	VAR robtarget OpenholeUD_2058 := [[509.33, -12.3, 177.5], [0.183051, 0.683002, 0.683002, -0.183051], [0,0,0,0], [9E9, 9E9, 9E9, 9E9, 9E9, 9E9]];
	VAR robtarget OpenholeUD_2059 := [[505.34, -12.3, 177.76], [0.154444, 0.690034, 0.680633, -0.191674], [0,0,0,0], [9E9, 9E9, 9E9, 9E9, 9E9, 9E9]];
	VAR robtarget OpenholeUD_2060 := [[501.35, -12.3, 178.01], [0.143713, 0.692349, 0.68338, -0.181638], [0,0,0,0], [9E9, 9E9, 9E9, 9E9, 9E9, 9E9]];
	VAR robtarget OpenholeUD_2061 := [[497.36, -12.3, 178.27], [0.132627, 0.694557, 0.686061, -0.17123], [0,0,0,0], [9E9, 9E9, 9E9, 9E9, 9E9, 9E9]];
	VAR robtarget OpenholeUD_2062 := [[493.37, -12.3, 178.53], [0.121195, 0.696643, 0.688661, -0.160454], [0,0,0,0], [9E9, 9E9, 9E9, 9E9, 9E9, 9E9]];
	VAR robtarget OpenholeUD_2063 := [[489.38, -12.3, 178.79], [0.109428, 0.698588, 0.691162, -0.149315], [0,0,0,0], [9E9, 9E9, 9E9, 9E9, 9E9, 9E9]];
	VAR robtarget OpenholeUD_2064 := [[485.38, -12.3, 179.05], [0.097343, 0.700374, 0.693545, -0.137825], [0,0,0,0], [9E9, 9E9, 9E9, 9E9, 9E9, 9E9]];
	VAR robtarget OpenholeUD_2065 := [[481.39, -12.3, 179.31], [0.084958, 0.701984, 0.695791, -0.125996], [0,0,0,0], [9E9, 9E9, 9E9, 9E9, 9E9, 9E9]];
	VAR robtarget OpenholeUD_2066 := [[477.4, -12.3, 179.56], [0.072297, 0.703401, 0.697881, -0.113848], [0,0,0,0], [9E9, 9E9, 9E9, 9E9, 9E9, 9E9]];
	VAR robtarget OpenholeUD_2067 := [[473.41, -12.3, 179.82], [0.059389, 0.704608, 0.699798, -0.101403], [0,0,0,0], [9E9, 9E9, 9E9, 9E9, 9E9, 9E9]];
	VAR robtarget OpenholeUD_2068 := [[469.42, -12.3, 180.08], [0.046265, 0.705592, 0.701523, -0.088688], [0,0,0,0], [9E9, 9E9, 9E9, 9E9, 9E9, 9E9]];
	VAR robtarget OpenholeUD_2069 := [[465.43, -12.3, 180.34], [0.032962, 0.706338, 0.703039, -0.075734], [0,0,0,0], [9E9, 9E9, 9E9, 9E9, 9E9, 9E9]];
	VAR robtarget OpenholeUD_2070 := [[461.43, -12.3, 180.6], [0.019518, 0.706837, 0.704333, -0.062574], [0,0,0,0], [9E9, 9E9, 9E9, 9E9, 9E9, 9E9]];
	VAR robtarget OpenholeUD_2071 := [[457.44, -12.3, 180.86], [0.005975, 0.707082, 0.70539, -0.049249], [0,0,0,0], [9E9, 9E9, 9E9, 9E9, 9E9, 9E9]];
	VAR robtarget OpenholeUD_2072 := [[453.45, -12.3, 181.12], [-0.007623, 0.707066, 0.7062, -0.035797], [0,0,0,0], [9E9, 9E9, 9E9, 9E9, 9E9, 9E9]];
	VAR robtarget OpenholeUD_2073 := [[449.46, -12.3, 181.37], [-0.021231, 0.706788, 0.706756, -0.022263], [0,0,0,0], [9E9, 9E9, 9E9, 9E9, 9E9, 9E9]];
	VAR robtarget OpenholeUD_2074 := [[445.47, -12.3, 181.63], [-0.034805, 0.70625, 0.707053, -0.008691], [0,0,0,0], [9E9, 9E9, 9E9, 9E9, 9E9, 9E9]];
	VAR robtarget OpenholeUD_2075 := [[441.48, -12.3, 181.89], [-0.048298, 0.705455, 0.70709, 0.004875], [0,0,0,0], [9E9, 9E9, 9E9, 9E9, 9E9, 9E9]];
	VAR robtarget OpenholeUD_2076 := [[437.48, -12.3, 182.15], [-0.061667, 0.704413, 0.706868, 0.01839], [0,0,0,0], [9E9, 9E9, 9E9, 9E9, 9E9, 9E9]];
	VAR robtarget OpenholeUD_2077 := [[433.49, -12.3, 182.41], [-0.074872, 0.703132, 0.706391, 0.03181], [0,0,0,0], [9E9, 9E9, 9E9, 9E9, 9E9, 9E9]];
	VAR robtarget OpenholeUD_2078 := [[429.5, -12.3, 182.67], [-0.087873, 0.701626, 0.705667, 0.045095], [0,0,0,0], [9E9, 9E9, 9E9, 9E9, 9E9, 9E9]];
	VAR robtarget OpenholeUD_2079 := [[425.51, -12.3, 182.92], [-0.100635, 0.699909, 0.704707, 0.058204], [0,0,0,0], [9E9, 9E9, 9E9, 9E9, 9E9, 9E9]];
	VAR robtarget OpenholeUD_2080 := [[421.52, -12.3, 183.18], [-0.113126, 0.697999, 0.703523, 0.071103], [0,0,0,0], [9E9, 9E9, 9E9, 9E9, 9E9, 9E9]];
	VAR robtarget OpenholeUD_2081 := [[417.53, -12.3, 183.44], [-0.125319, 0.695913, 0.702128, 0.08376], [0,0,0,0], [9E9, 9E9, 9E9, 9E9, 9E9, 9E9]];
	VAR robtarget OpenholeUD_2082 := [[413.54, -12.3, 183.7], [-0.137192, 0.69367, 0.70054, 0.096145], [0,0,0,0], [9E9, 9E9, 9E9, 9E9, 9E9, 9E9]];
	VAR robtarget OpenholeUD_2083 := [[409.54, -12.3, 183.96], [-0.148726, 0.691289, 0.698774, 0.108235], [0,0,0,0], [9E9, 9E9, 9E9, 9E9, 9E9, 9E9]];
	VAR robtarget OpenholeUD_2084 := [[405.55, -12.3, 184.22], [-0.159905, 0.688789, 0.696848, 0.120011], [0,0,0,0], [9E9, 9E9, 9E9, 9E9, 9E9, 9E9]];
	VAR robtarget OpenholeUD_2085 := [[401.56, -12.3, 184.48], [-0.170721, 0.686188, 0.69478, 0.131455], [0,0,0,0], [9E9, 9E9, 9E9, 9E9, 9E9, 9E9]];
	VAR robtarget OpenholeUD_2086 := [[397.57, -12.3, 184.73], [-0.181166, 0.683505, 0.692588, 0.142556], [0,0,0,0], [9E9, 9E9, 9E9, 9E9, 9E9, 9E9]];
	VAR robtarget OpenholeUD_2087 := [[393.58, -12.3, 184.99], [-0.191237, 0.680756, 0.690288, 0.153306], [0,0,0,0], [9E9, 9E9, 9E9, 9E9, 9E9, 9E9]];
	VAR robtarget OpenholeUD_2088 := [[389.36, -12.3, 185.27], [-0.201475, 0.677796, 0.687759, 0.164279], [0,0,0,0], [9E9, 9E9, 9E9, 9E9, 9E9, 9E9]];
	VAR robtarget OpenholeUD_2089 := [[385.36, -12.3, 185.28], [-0.183051, 0.683002, 0.683002, 0.183051], [0,0,0,0], [9E9, 9E9, 9E9, 9E9, 9E9, 9E9]];
	VAR robtarget OpenholeUD_2090 := [[381.36, -12.3, 185.29], [-0.183051, 0.683002, 0.683002, 0.183051], [0,0,0,0], [9E9, 9E9, 9E9, 9E9, 9E9, 9E9]];
	VAR robtarget OpenholeUD_2091 := [[377.36, -12.3, 185.3], [-0.183051, 0.683002, 0.683002, 0.183051], [0,0,0,0], [9E9, 9E9, 9E9, 9E9, 9E9, 9E9]];
	VAR robtarget OpenholeUD_2092 := [[373.36, -12.3, 185.32], [-0.183051, 0.683002, 0.683002, 0.183051], [0,0,0,0], [9E9, 9E9, 9E9, 9E9, 9E9, 9E9]];
	VAR robtarget OpenholeUD_2093 := [[369.36, -12.3, 185.33], [-0.183051, 0.683002, 0.683002, 0.183051], [0,0,0,0], [9E9, 9E9, 9E9, 9E9, 9E9, 9E9]];
	VAR robtarget OpenholeUD_2094 := [[369.36, -12.3, 185.33], [-0.183051, 0.683002, 0.683002, 0.183051], [0,0,0,0], [9E9, 9E9, 9E9, 9E9, 9E9, 9E9]];
	VAR robtarget OpenholeUD_2095 := [[369.36, -13.5, 184.64], [-0.183051, 0.683002, 0.683002, 0.183051], [0,0,0,0], [9E9, 9E9, 9E9, 9E9, 9E9, 9E9]];
	VAR robtarget OpenholeUD_2096 := [[373.36, -13.5, 184.62], [-0.183051, 0.683002, 0.683002, 0.183051], [0,0,0,0], [9E9, 9E9, 9E9, 9E9, 9E9, 9E9]];
	VAR robtarget OpenholeUD_2097 := [[377.36, -13.5, 184.61], [-0.183051, 0.683002, 0.683002, 0.183051], [0,0,0,0], [9E9, 9E9, 9E9, 9E9, 9E9, 9E9]];
	VAR robtarget OpenholeUD_2098 := [[381.36, -13.5, 184.6], [-0.183051, 0.683002, 0.683002, 0.183051], [0,0,0,0], [9E9, 9E9, 9E9, 9E9, 9E9, 9E9]];
	VAR robtarget OpenholeUD_2099 := [[385.36, -13.5, 184.59], [-0.183051, 0.683002, 0.683002, 0.183051], [0,0,0,0], [9E9, 9E9, 9E9, 9E9, 9E9, 9E9]];
	VAR robtarget OpenholeUD_2100 := [[389.36, -13.5, 184.57], [-0.198088, 0.678794, 0.686931, 0.167708], [0,0,0,0], [9E9, 9E9, 9E9, 9E9, 9E9, 9E9]];
	VAR robtarget OpenholeUD_2101 := [[393.35, -13.5, 184.36], [-0.188336, 0.681564, 0.689367, 0.157396], [0,0,0,0], [9E9, 9E9, 9E9, 9E9, 9E9, 9E9]];
	VAR robtarget OpenholeUD_2102 := [[397.34, -13.5, 184.15], [-0.17821, 0.684281, 0.691716, 0.146726], [0,0,0,0], [9E9, 9E9, 9E9, 9E9, 9E9, 9E9]];
	VAR robtarget OpenholeUD_2103 := [[401.34, -13.5, 183.94], [-0.167712, 0.68693, 0.693963, 0.135702], [0,0,0,0], [9E9, 9E9, 9E9, 9E9, 9E9, 9E9]];
	VAR robtarget OpenholeUD_2104 := [[405.33, -13.5, 183.72], [-0.156844, 0.689493, 0.69609, 0.124331], [0,0,0,0], [9E9, 9E9, 9E9, 9E9, 9E9, 9E9]];
	VAR robtarget OpenholeUD_2105 := [[409.33, -13.5, 183.51], [-0.145614, 0.691951, 0.69808, 0.112626], [0,0,0,0], [9E9, 9E9, 9E9, 9E9, 9E9, 9E9]];
	VAR robtarget OpenholeUD_2106 := [[413.32, -13.5, 183.3], [-0.134032, 0.694288, 0.699914, 0.1006], [0,0,0,0], [9E9, 9E9, 9E9, 9E9, 9E9, 9E9]];
	VAR robtarget OpenholeUD_2107 := [[417.32, -13.5, 183.09], [-0.122114, 0.696483, 0.701575, 0.088273], [0,0,0,0], [9E9, 9E9, 9E9, 9E9, 9E9, 9E9]];
	VAR robtarget OpenholeUD_2108 := [[421.31, -13.5, 182.87], [-0.109878, 0.698518, 0.703046, 0.07567], [0,0,0,0], [9E9, 9E9, 9E9, 9E9, 9E9, 9E9]];
	VAR robtarget OpenholeUD_2109 := [[425.31, -13.5, 182.66], [-0.097347, 0.700374, 0.704311, 0.062816], [0,0,0,0], [9E9, 9E9, 9E9, 9E9, 9E9, 9E9]];
	VAR robtarget OpenholeUD_2110 := [[429.3, -13.5, 182.45], [-0.08455, 0.702034, 0.705355, 0.049744], [0,0,0,0], [9E9, 9E9, 9E9, 9E9, 9E9, 9E9]];
	VAR robtarget OpenholeUD_2111 := [[433.29, -13.5, 182.24], [-0.071518, 0.703481, 0.706165, 0.036489], [0,0,0,0], [9E9, 9E9, 9E9, 9E9, 9E9, 9E9]];
	VAR robtarget OpenholeUD_2112 := [[437.29, -13.5, 182.02], [-0.058286, 0.7047, 0.70673, 0.023089], [0,0,0,0], [9E9, 9E9, 9E9, 9E9, 9E9, 9E9]];
	VAR robtarget OpenholeUD_2113 := [[441.28, -13.5, 181.81], [-0.044894, 0.70568, 0.707042, 0.009586], [0,0,0,0], [9E9, 9E9, 9E9, 9E9, 9E9, 9E9]];
	VAR robtarget OpenholeUD_2114 := [[445.45, -13.5, 181.59], [-0.030809, 0.706435, 0.707092, -0.004555], [0,0,0,0], [9E9, 9E9, 9E9, 9E9, 9E9, 9E9]];
	VAR robtarget OpenholeUD_2115 := [[445.45, -13.5, 181.59], [-0.030809, 0.706435, 0.707092, -0.004555], [0,0,0,0], [9E9, 9E9, 9E9, 9E9, 9E9, 9E9]];
	VAR robtarget OpenholeUD_2116 := [[444.22, -14.7, 181.59], [-0.030884, 0.706432, 0.707097, 0.003667], [0,0,0,0], [9E9, 9E9, 9E9, 9E9, 9E9, 9E9]];
	VAR robtarget OpenholeUD_2117 := [[440.23, -14.7, 181.76], [-0.04439, 0.705712, 0.706897, 0.017215], [0,0,0,0], [9E9, 9E9, 9E9, 9E9, 9E9, 9E9]];
	VAR robtarget OpenholeUD_2118 := [[436.23, -14.7, 181.93], [-0.057772, 0.704743, 0.706441, 0.030684], [0,0,0,0], [9E9, 9E9, 9E9, 9E9, 9E9, 9E9]];
	VAR robtarget OpenholeUD_2119 := [[432.23, -14.7, 182.09], [-0.07099, 0.703534, 0.705735, 0.04403], [0,0,0,0], [9E9, 9E9, 9E9, 9E9, 9E9, 9E9]];
	VAR robtarget OpenholeUD_2120 := [[428.24, -14.7, 182.26], [-0.084005, 0.702099, 0.704788, 0.057215], [0,0,0,0], [9E9, 9E9, 9E9, 9E9, 9E9, 9E9]];
	VAR robtarget OpenholeUD_2121 := [[424.24, -14.7, 182.43], [-0.096783, 0.700452, 0.703613, 0.070201], [0,0,0,0], [9E9, 9E9, 9E9, 9E9, 9E9, 9E9]];
	VAR robtarget OpenholeUD_2122 := [[420.24, -14.7, 182.59], [-0.109291, 0.69861, 0.702224, 0.082953], [0,0,0,0], [9E9, 9E9, 9E9, 9E9, 9E9, 9E9]];
	VAR robtarget OpenholeUD_2123 := [[416.25, -14.7, 182.76], [-0.121503, 0.69659, 0.700636, 0.095443], [0,0,0,0], [9E9, 9E9, 9E9, 9E9, 9E9, 9E9]];
	VAR robtarget OpenholeUD_2124 := [[412.25, -14.7, 182.93], [-0.133395, 0.69441, 0.698865, 0.107643], [0,0,0,0], [9E9, 9E9, 9E9, 9E9, 9E9, 9E9]];
	VAR robtarget OpenholeUD_2125 := [[408.25, -14.7, 183.09], [-0.14495, 0.692091, 0.69693, 0.119534], [0,0,0,0], [9E9, 9E9, 9E9, 9E9, 9E9, 9E9]];
	VAR robtarget OpenholeUD_2126 := [[404.26, -14.7, 183.26], [-0.156153, 0.689649, 0.694848, 0.131096], [0,0,0,0], [9E9, 9E9, 9E9, 9E9, 9E9, 9E9]];
	VAR robtarget OpenholeUD_2127 := [[400.26, -14.7, 183.43], [-0.166993, 0.687105, 0.692637, 0.142317], [0,0,0,0], [9E9, 9E9, 9E9, 9E9, 9E9, 9E9]];
	VAR robtarget OpenholeUD_2128 := [[396.27, -14.7, 183.59], [-0.177464, 0.684475, 0.690315, 0.153186], [0,0,0,0], [9E9, 9E9, 9E9, 9E9, 9E9, 9E9]];
	VAR robtarget OpenholeUD_2129 := [[389.35, -14.7, 183.88], [-0.194694, 0.679775, 0.686085, 0.171135], [0,0,0,0], [9E9, 9E9, 9E9, 9E9, 9E9, 9E9]];
	VAR robtarget OpenholeUD_2130 := [[385.35, -14.7, 183.89], [-0.183051, 0.683002, 0.683002, 0.183051], [0,0,0,0], [9E9, 9E9, 9E9, 9E9, 9E9, 9E9]];
	VAR robtarget OpenholeUD_2131 := [[381.35, -14.7, 183.91], [-0.183051, 0.683002, 0.683002, 0.183051], [0,0,0,0], [9E9, 9E9, 9E9, 9E9, 9E9, 9E9]];
	VAR robtarget OpenholeUD_2132 := [[377.35, -14.7, 183.92], [-0.183051, 0.683002, 0.683002, 0.183051], [0,0,0,0], [9E9, 9E9, 9E9, 9E9, 9E9, 9E9]];
	VAR robtarget OpenholeUD_2133 := [[369.35, -14.7, 183.94], [-0.183051, 0.683002, 0.683002, 0.183051], [0,0,0,0], [9E9, 9E9, 9E9, 9E9, 9E9, 9E9]];
	VAR robtarget OpenholeUD_2134 := [[369.35, -14.7, 183.94], [-0.183051, 0.683002, 0.683002, 0.183051], [0,0,0,0], [9E9, 9E9, 9E9, 9E9, 9E9, 9E9]];
	VAR robtarget OpenholeUD_2135 := [[369.35, -15.9, 183.25], [-0.183051, 0.683002, 0.683002, 0.183051], [0,0,0,0], [9E9, 9E9, 9E9, 9E9, 9E9, 9E9]];
	VAR robtarget OpenholeUD_2136 := [[373.35, -15.9, 183.24], [-0.183051, 0.683002, 0.683002, 0.183051], [0,0,0,0], [9E9, 9E9, 9E9, 9E9, 9E9, 9E9]];
	VAR robtarget OpenholeUD_2137 := [[377.35, -15.9, 183.22], [-0.183051, 0.683002, 0.683002, 0.183051], [0,0,0,0], [9E9, 9E9, 9E9, 9E9, 9E9, 9E9]];
	VAR robtarget OpenholeUD_2138 := [[381.35, -15.9, 183.21], [-0.183051, 0.683002, 0.683002, 0.183051], [0,0,0,0], [9E9, 9E9, 9E9, 9E9, 9E9, 9E9]];
	VAR robtarget OpenholeUD_2139 := [[389.35, -15.9, 183.19], [-0.191292, 0.68074, 0.685222, 0.174561], [0,0,0,0], [9E9, 9E9, 9E9, 9E9, 9E9, 9E9]];
	VAR robtarget OpenholeUD_2140 := [[393.35, -15.9, 183.07], [-0.181391, 0.683445, 0.687735, 0.164377], [0,0,0,0], [9E9, 9E9, 9E9, 9E9, 9E9, 9E9]];
	VAR robtarget OpenholeUD_2141 := [[397.35, -15.9, 182.95], [-0.171117, 0.68609, 0.690171, 0.153832], [0,0,0,0], [9E9, 9E9, 9E9, 9E9, 9E9, 9E9]];
	VAR robtarget OpenholeUD_2142 := [[401.35, -15.9, 182.83], [-0.160474, 0.688657, 0.692511, 0.142928], [0,0,0,0], [9E9, 9E9, 9E9, 9E9, 9E9, 9E9]];
	VAR robtarget OpenholeUD_2143 := [[405.34, -15.9, 182.71], [-0.149465, 0.69113, 0.694739, 0.131672], [0,0,0,0], [9E9, 9E9, 9E9, 9E9, 9E9, 9E9]];
	VAR robtarget OpenholeUD_2144 := [[409.34, -15.9, 182.59], [-0.138098, 0.69349, 0.696837, 0.120075], [0,0,0,0], [9E9, 9E9, 9E9, 9E9, 9E9, 9E9]];
	VAR robtarget OpenholeUD_2145 := [[413.34, -15.9, 182.46], [-0.126386, 0.69572, 0.698787, 0.108151], [0,0,0,0], [9E9, 9E9, 9E9, 9E9, 9E9, 9E9]];
	VAR robtarget OpenholeUD_2146 := [[417.34, -15.9, 182.34], [-0.114345, 0.6978, 0.700571, 0.095917], [0,0,0,0], [9E9, 9E9, 9E9, 9E9, 9E9, 9E9]];
	VAR robtarget OpenholeUD_2147 := [[421.34, -15.9, 182.22], [-0.101994, 0.699712, 0.702172, 0.083396], [0,0,0,0], [9E9, 9E9, 9E9, 9E9, 9E9, 9E9]];
	VAR robtarget OpenholeUD_2148 := [[425.34, -15.9, 182.1], [-0.089359, 0.701438, 0.703572, 0.070615], [0,0,0,0], [9E9, 9E9, 9E9, 9E9, 9E9, 9E9]];
	VAR robtarget OpenholeUD_2149 := [[429.33, -15.9, 181.98], [-0.076469, 0.70296, 0.704757, 0.057603], [0,0,0,0], [9E9, 9E9, 9E9, 9E9, 9E9, 9E9]];
	VAR robtarget OpenholeUD_2150 := [[433.33, -15.9, 181.86], [-0.063356, 0.704263, 0.705712, 0.044396], [0,0,0,0], [9E9, 9E9, 9E9, 9E9, 9E9, 9E9]];
	VAR robtarget OpenholeUD_2151 := [[437.33, -15.9, 181.74], [-0.050056, 0.705333, 0.706426, 0.031031], [0,0,0,0], [9E9, 9E9, 9E9, 9E9, 9E9, 9E9]];
	VAR robtarget OpenholeUD_2152 := [[443.48, -15.9, 181.56], [-0.029327, 0.706498, 0.707032, 0.010255], [0,0,0,0], [9E9, 9E9, 9E9, 9E9, 9E9, 9E9]];
	VAR robtarget OpenholeUD_2153 := [[443.48, -15.9, 181.56], [-0.029327, 0.706498, 0.707032, 0.010255], [0,0,0,0], [9E9, 9E9, 9E9, 9E9, 9E9, 9E9]];
	VAR robtarget OpenholeUD_2154 := [[443.05, -17.1, 181.5], [-0.026721, 0.706602, 0.70693, 0.015795], [0,0,0,0], [9E9, 9E9, 9E9, 9E9, 9E9, 9E9]];
	VAR robtarget OpenholeUD_2155 := [[439.05, -17.1, 181.57], [-0.040236, 0.705961, 0.706499, 0.029304], [0,0,0,0], [9E9, 9E9, 9E9, 9E9, 9E9, 9E9]];
	VAR robtarget OpenholeUD_2156 := [[435.05, -17.1, 181.65], [-0.053629, 0.70507, 0.705816, 0.042707], [0,0,0,0], [9E9, 9E9, 9E9, 9E9, 9E9, 9E9]];
	VAR robtarget OpenholeUD_2157 := [[431.05, -17.1, 181.72], [-0.066861, 0.703939, 0.704889, 0.055961], [0,0,0,0], [9E9, 9E9, 9E9, 9E9, 9E9, 9E9]];
	VAR robtarget OpenholeUD_2158 := [[427.05, -17.1, 181.79], [-0.079891, 0.702579, 0.703729, 0.069029], [0,0,0,0], [9E9, 9E9, 9E9, 9E9, 9E9, 9E9]];
	VAR robtarget OpenholeUD_2159 := [[423.05, -17.1, 181.87], [-0.092685, 0.701006, 0.702351, 0.081875], [0,0,0,0], [9E9, 9E9, 9E9, 9E9, 9E9, 9E9]];
	VAR robtarget OpenholeUD_2160 := [[419.05, -17.1, 181.94], [-0.105212, 0.699236, 0.700768, 0.094468], [0,0,0,0], [9E9, 9E9, 9E9, 9E9, 9E9, 9E9]];
	VAR robtarget OpenholeUD_2161 := [[415.05, -17.1, 182.02], [-0.117445, 0.697285, 0.698998, 0.106779], [0,0,0,0], [9E9, 9E9, 9E9, 9E9, 9E9, 9E9]];
	VAR robtarget OpenholeUD_2162 := [[411.05, -17.1, 182.09], [-0.12936, 0.695173, 0.697058, 0.118786], [0,0,0,0], [9E9, 9E9, 9E9, 9E9, 9E9, 9E9]];
	VAR robtarget OpenholeUD_2163 := [[407.05, -17.1, 182.17], [-0.14094, 0.692918, 0.694966, 0.130469], [0,0,0,0], [9E9, 9E9, 9E9, 9E9, 9E9, 9E9]];
	VAR robtarget OpenholeUD_2164 := [[403.05, -17.1, 182.24], [-0.15217, 0.690539, 0.69274, 0.141813], [0,0,0,0], [9E9, 9E9, 9E9, 9E9, 9E9, 9E9]];
	VAR robtarget OpenholeUD_2165 := [[399.05, -17.1, 182.31], [-0.163039, 0.688054, 0.690399, 0.152806], [0,0,0,0], [9E9, 9E9, 9E9, 9E9, 9E9, 9E9]];
	VAR robtarget OpenholeUD_2166 := [[395.06, -17.1, 182.39], [-0.173542, 0.68548, 0.687959, 0.16344], [0,0,0,0], [9E9, 9E9, 9E9, 9E9, 9E9, 9E9]];
	VAR robtarget OpenholeUD_2167 := [[389.35, -17.1, 182.49], [-0.187884, 0.681689, 0.68434, 0.177984], [0,0,0,0], [9E9, 9E9, 9E9, 9E9, 9E9, 9E9]];
	VAR robtarget OpenholeUD_2168 := [[385.35, -17.1, 182.51], [-0.183051, 0.683002, 0.683002, 0.183051], [0,0,0,0], [9E9, 9E9, 9E9, 9E9, 9E9, 9E9]];
	VAR robtarget OpenholeUD_2169 := [[381.35, -17.1, 182.52], [-0.183051, 0.683002, 0.683002, 0.183051], [0,0,0,0], [9E9, 9E9, 9E9, 9E9, 9E9, 9E9]];
	VAR robtarget OpenholeUD_2170 := [[377.35, -17.1, 182.53], [-0.183051, 0.683002, 0.683002, 0.183051], [0,0,0,0], [9E9, 9E9, 9E9, 9E9, 9E9, 9E9]];
	VAR robtarget OpenholeUD_2171 := [[369.35, -17.1, 182.56], [-0.183051, 0.683002, 0.683002, 0.183051], [0,0,0,0], [9E9, 9E9, 9E9, 9E9, 9E9, 9E9]];
	VAR robtarget OpenholeUD_2172 := [[369.35, -17.1, 182.56], [-0.183051, 0.683002, 0.683002, 0.183051], [0,0,0,0], [9E9, 9E9, 9E9, 9E9, 9E9, 9E9]];
	VAR robtarget OpenholeUD_2173 := [[369.35, -18.3, 181.86], [-0.183051, 0.683002, 0.683002, 0.183051], [0,0,0,0], [9E9, 9E9, 9E9, 9E9, 9E9, 9E9]];
	VAR robtarget OpenholeUD_2174 := [[373.35, -18.3, 181.85], [-0.183051, 0.683002, 0.683002, 0.183051], [0,0,0,0], [9E9, 9E9, 9E9, 9E9, 9E9, 9E9]];
	VAR robtarget OpenholeUD_2175 := [[377.35, -18.3, 181.84], [-0.183051, 0.683002, 0.683002, 0.183051], [0,0,0,0], [9E9, 9E9, 9E9, 9E9, 9E9, 9E9]];
	VAR robtarget OpenholeUD_2176 := [[381.35, -18.3, 181.83], [-0.183051, 0.683002, 0.683002, 0.183051], [0,0,0,0], [9E9, 9E9, 9E9, 9E9, 9E9, 9E9]];
	VAR robtarget OpenholeUD_2177 := [[385.35, -18.3, 181.81], [-0.183051, 0.683002, 0.683002, 0.183051], [0,0,0,0], [9E9, 9E9, 9E9, 9E9, 9E9, 9E9]];
	VAR robtarget OpenholeUD_2178 := [[389.35, -18.3, 181.8], [-0.18447, 0.682621, 0.683442, 0.181403], [0,0,0,0], [9E9, 9E9, 9E9, 9E9, 9E9, 9E9]];
	VAR robtarget OpenholeUD_2179 := [[393.35, -18.3, 181.77], [-0.174424, 0.685256, 0.68603, 0.171354], [0,0,0,0], [9E9, 9E9, 9E9, 9E9, 9E9, 9E9]];
	VAR robtarget OpenholeUD_2180 := [[397.35, -18.3, 181.74], [-0.164009, 0.687823, 0.688548, 0.160941], [0,0,0,0], [9E9, 9E9, 9E9, 9E9, 9E9, 9E9]];
	VAR robtarget OpenholeUD_2181 := [[401.35, -18.3, 181.72], [-0.153227, 0.690305, 0.690978, 0.150165], [0,0,0,0], [9E9, 9E9, 9E9, 9E9, 9E9, 9E9]];
	VAR robtarget OpenholeUD_2182 := [[405.35, -18.3, 181.69], [-0.142084, 0.692685, 0.693304, 0.139032], [0,0,0,0], [9E9, 9E9, 9E9, 9E9, 9E9, 9E9]];
	VAR robtarget OpenholeUD_2183 := [[409.35, -18.3, 181.66], [-0.130588, 0.694944, 0.695507, 0.127552], [0,0,0,0], [9E9, 9E9, 9E9, 9E9, 9E9, 9E9]];
	VAR robtarget OpenholeUD_2184 := [[413.35, -18.3, 181.63], [-0.118754, 0.697064, 0.697571, 0.115737], [0,0,0,0], [9E9, 9E9, 9E9, 9E9, 9E9, 9E9]];
	VAR robtarget OpenholeUD_2185 := [[417.35, -18.3, 181.61], [-0.106598, 0.699026, 0.699476, 0.103605], [0,0,0,0], [9E9, 9E9, 9E9, 9E9, 9E9, 9E9]];
	VAR robtarget OpenholeUD_2186 := [[421.35, -18.3, 181.58], [-0.094141, 0.700812, 0.701204, 0.091176], [0,0,0,0], [9E9, 9E9, 9E9, 9E9, 9E9, 9E9]];
	VAR robtarget OpenholeUD_2187 := [[425.35, -18.3, 181.55], [-0.081411, 0.702405, 0.702739, 0.078477], [0,0,0,0], [9E9, 9E9, 9E9, 9E9, 9E9, 9E9]];
	VAR robtarget OpenholeUD_2188 := [[429.35, -18.3, 181.52], [-0.068436, 0.703787, 0.704063, 0.065535], [0,0,0,0], [9E9, 9E9, 9E9, 9E9, 9E9, 9E9]];
	VAR robtarget OpenholeUD_2189 := [[433.35, -18.3, 181.49], [-0.055252, 0.704945, 0.705164, 0.052386], [0,0,0,0], [9E9, 9E9, 9E9, 9E9, 9E9, 9E9]];
	VAR robtarget OpenholeUD_2190 := [[437.35, -18.3, 181.47], [-0.041895, 0.705865, 0.706027, 0.039065], [0,0,0,0], [9E9, 9E9, 9E9, 9E9, 9E9, 9E9]];
	VAR robtarget OpenholeUD_2191 := [[442.86, -18.3, 181.43], [-0.023279, 0.706723, 0.70681, 0.0205], [0,0,0,0], [9E9, 9E9, 9E9, 9E9, 9E9, 9E9]];
	VAR robtarget OpenholeUD_2192 := [[442.86, -18.3, 181.43], [-0.023279, 0.706723, 0.70681, 0.0205], [0,0,0,0], [9E9, 9E9, 9E9, 9E9, 9E9, 9E9]];
	VAR robtarget OpenholeUD_2193 := [[442.9, -19.5, 181.35], [-0.019074, 0.706849, 0.706684, 0.024443], [0,0,0,0], [9E9, 9E9, 9E9, 9E9, 9E9, 9E9]];
	VAR robtarget OpenholeUD_2194 := [[438.9, -19.5, 181.33], [-0.032618, 0.706354, 0.706089, 0.037919], [0,0,0,0], [9E9, 9E9, 9E9, 9E9, 9E9, 9E9]];
	VAR robtarget OpenholeUD_2195 := [[434.9, -19.5, 181.32], [-0.046054, 0.705605, 0.705245, 0.051273], [0,0,0,0], [9E9, 9E9, 9E9, 9E9, 9E9, 9E9]];
	VAR robtarget OpenholeUD_2196 := [[430.9, -19.5, 181.3], [-0.059339, 0.704613, 0.704162, 0.064463], [0,0,0,0], [9E9, 9E9, 9E9, 9E9, 9E9, 9E9]];
	VAR robtarget OpenholeUD_2197 := [[426.9, -19.5, 181.28], [-0.072435, 0.703387, 0.702852, 0.077453], [0,0,0,0], [9E9, 9E9, 9E9, 9E9, 9E9, 9E9]];
	VAR robtarget OpenholeUD_2198 := [[422.9, -19.5, 181.26], [-0.085306, 0.701942, 0.701329, 0.090208], [0,0,0,0], [9E9, 9E9, 9E9, 9E9, 9E9, 9E9]];
	VAR robtarget OpenholeUD_2199 := [[418.9, -19.5, 181.24], [-0.09792, 0.700294, 0.699609, 0.102697], [0,0,0,0], [9E9, 9E9, 9E9, 9E9, 9E9, 9E9]];
	VAR robtarget OpenholeUD_2200 := [[414.9, -19.5, 181.22], [-0.110247, 0.698459, 0.69771, 0.114895], [0,0,0,0], [9E9, 9E9, 9E9, 9E9, 9E9, 9E9]];
	VAR robtarget OpenholeUD_2201 := [[410.9, -19.5, 181.21], [-0.122265, 0.696456, 0.695649, 0.126778], [0,0,0,0], [9E9, 9E9, 9E9, 9E9, 9E9, 9E9]];
	VAR robtarget OpenholeUD_2202 := [[406.9, -19.5, 181.19], [-0.133955, 0.694303, 0.693444, 0.138329], [0,0,0,0], [9E9, 9E9, 9E9, 9E9, 9E9, 9E9]];
	VAR robtarget OpenholeUD_2203 := [[402.9, -19.5, 181.17], [-0.145299, 0.692017, 0.691115, 0.149535], [0,0,0,0], [9E9, 9E9, 9E9, 9E9, 9E9, 9E9]];
	VAR robtarget OpenholeUD_2204 := [[398.9, -19.5, 181.15], [-0.156289, 0.689619, 0.688678, 0.160384], [0,0,0,0], [9E9, 9E9, 9E9, 9E9, 9E9, 9E9]];
	VAR robtarget OpenholeUD_2205 := [[394.9, -19.5, 181.13], [-0.166914, 0.687124, 0.686151, 0.170871], [0,0,0,0], [9E9, 9E9, 9E9, 9E9, 9E9, 9E9]];
	VAR robtarget OpenholeUD_2206 := [[389.35, -19.5, 181.11], [-0.181051, 0.683535, 0.682526, 0.184819], [0,0,0,0], [9E9, 9E9, 9E9, 9E9, 9E9, 9E9]];
	VAR robtarget OpenholeUD_2207 := [[385.35, -19.5, 181.12], [-0.183051, 0.683002, 0.683002, 0.183051], [0,0,0,0], [9E9, 9E9, 9E9, 9E9, 9E9, 9E9]];
	VAR robtarget OpenholeUD_2208 := [[381.35, -19.5, 181.13], [-0.183051, 0.683002, 0.683002, 0.183051], [0,0,0,0], [9E9, 9E9, 9E9, 9E9, 9E9, 9E9]];
	VAR robtarget OpenholeUD_2209 := [[377.35, -19.5, 181.15], [-0.183051, 0.683002, 0.683002, 0.183051], [0,0,0,0], [9E9, 9E9, 9E9, 9E9, 9E9, 9E9]];
	VAR robtarget OpenholeUD_2210 := [[373.35, -19.5, 181.16], [-0.183051, 0.683002, 0.683002, 0.183051], [0,0,0,0], [9E9, 9E9, 9E9, 9E9, 9E9, 9E9]];
	VAR robtarget OpenholeUD_2211 := [[369.35, -19.5, 181.17], [-0.183051, 0.683002, 0.683002, 0.183051], [0,0,0,0], [9E9, 9E9, 9E9, 9E9, 9E9, 9E9]];
	VAR robtarget OpenholeUD_2212 := [[369.35, -19.5, 181.17], [-0.183051, 0.683002, 0.683002, 0.183051], [0,0,0,0], [9E9, 9E9, 9E9, 9E9, 9E9, 9E9]];
	VAR robtarget OpenholeUD_2213 := [[369.34, -20.7, 180.48], [-0.183051, 0.683002, 0.683002, 0.183051], [0,0,0,0], [9E9, 9E9, 9E9, 9E9, 9E9, 9E9]];
	VAR robtarget OpenholeUD_2214 := [[373.34, -20.7, 180.47], [-0.183051, 0.683002, 0.683002, 0.183051], [0,0,0,0], [9E9, 9E9, 9E9, 9E9, 9E9, 9E9]];
	VAR robtarget OpenholeUD_2215 := [[377.34, -20.7, 180.45], [-0.183051, 0.683002, 0.683002, 0.183051], [0,0,0,0], [9E9, 9E9, 9E9, 9E9, 9E9, 9E9]];
	VAR robtarget OpenholeUD_2216 := [[381.34, -20.7, 180.44], [-0.183051, 0.683002, 0.683002, 0.183051], [0,0,0,0], [9E9, 9E9, 9E9, 9E9, 9E9, 9E9]];
	VAR robtarget OpenholeUD_2217 := [[385.34, -20.7, 180.43], [-0.183051, 0.683002, 0.683002, 0.183051], [0,0,0,0], [9E9, 9E9, 9E9, 9E9, 9E9, 9E9]];
	VAR robtarget OpenholeUD_2218 := [[389.34, -20.7, 180.41], [-0.177628, 0.684433, 0.681594, 0.188229], [0,0,0,0], [9E9, 9E9, 9E9, 9E9, 9E9, 9E9]];
	VAR robtarget OpenholeUD_2219 := [[393.34, -20.7, 180.48], [-0.167444, 0.686995, 0.684253, 0.178321], [0,0,0,0], [9E9, 9E9, 9E9, 9E9, 9E9, 9E9]];
	VAR robtarget OpenholeUD_2220 := [[397.34, -20.7, 180.54], [-0.156894, 0.689481, 0.686848, 0.168045], [0,0,0,0], [9E9, 9E9, 9E9, 9E9, 9E9, 9E9]];
	VAR robtarget OpenholeUD_2221 := [[401.34, -20.7, 180.61], [-0.14598, 0.691874, 0.689365, 0.157404], [0,0,0,0], [9E9, 9E9, 9E9, 9E9, 9E9, 9E9]];
	VAR robtarget OpenholeUD_2222 := [[405.34, -20.7, 180.67], [-0.134709, 0.694157, 0.691785, 0.146401], [0,0,0,0], [9E9, 9E9, 9E9, 9E9, 9E9, 9E9]];
	VAR robtarget OpenholeUD_2223 := [[409.34, -20.7, 180.74], [-0.123092, 0.69631, 0.694091, 0.135046], [0,0,0,0], [9E9, 9E9, 9E9, 9E9, 9E9, 9E9]];
	VAR robtarget OpenholeUD_2224 := [[413.34, -20.7, 180.8], [-0.111144, 0.698317, 0.696265, 0.12335], [0,0,0,0], [9E9, 9E9, 9E9, 9E9, 9E9, 9E9]];
	VAR robtarget OpenholeUD_2225 := [[417.34, -20.7, 180.87], [-0.098881, 0.700159, 0.698288, 0.111328], [0,0,0,0], [9E9, 9E9, 9E9, 9E9, 9E9, 9E9]];
	VAR robtarget OpenholeUD_2226 := [[421.34, -20.7, 180.93], [-0.086329, 0.701817, 0.700142, 0.099001], [0,0,0,0], [9E9, 9E9, 9E9, 9E9, 9E9, 9E9]];
	VAR robtarget OpenholeUD_2227 := [[425.34, -20.7, 180.99], [-0.073512, 0.703275, 0.701809, 0.086392], [0,0,0,0], [9E9, 9E9, 9E9, 9E9, 9E9, 9E9]];
	VAR robtarget OpenholeUD_2228 := [[429.34, -20.7, 181.06], [-0.060463, 0.704517, 0.703273, 0.073531], [0,0,0,0], [9E9, 9E9, 9E9, 9E9, 9E9, 9E9]];
	VAR robtarget OpenholeUD_2229 := [[433.34, -20.7, 181.12], [-0.047217, 0.705529, 0.704518, 0.060449], [0,0,0,0], [9E9, 9E9, 9E9, 9E9, 9E9, 9E9]];
	VAR robtarget OpenholeUD_2230 := [[437.34, -20.7, 181.19], [-0.033812, 0.706298, 0.705531, 0.047182], [0,0,0,0], [9E9, 9E9, 9E9, 9E9, 9E9, 9E9]];
	VAR robtarget OpenholeUD_2231 := [[443.16, -20.7, 181.28], [-0.014092, 0.706966, 0.706567, 0.027613], [0,0,0,0], [9E9, 9E9, 9E9, 9E9, 9E9, 9E9]];
	VAR robtarget OpenholeUD_2232 := [[443.16, -20.7, 181.28], [-0.014092, 0.706966, 0.706567, 0.027613], [0,0,0,0], [9E9, 9E9, 9E9, 9E9, 9E9, 9E9]];
	VAR robtarget OpenholeUD_2233 := [[443.69, -21.9, 181.22], [-0.00822, 0.707059, 0.706474, 0.029897], [0,0,0,0], [9E9, 9E9, 9E9, 9E9, 9E9, 9E9]];
	VAR robtarget OpenholeUD_2234 := [[439.69, -21.9, 181.11], [-0.021801, 0.706771, 0.705776, 0.043357], [0,0,0,0], [9E9, 9E9, 9E9, 9E9, 9E9, 9E9]];
	VAR robtarget OpenholeUD_2235 := [[435.69, -21.9, 181], [-0.035297, 0.706225, 0.704831, 0.056689], [0,0,0,0], [9E9, 9E9, 9E9, 9E9, 9E9, 9E9]];
	VAR robtarget OpenholeUD_2236 := [[431.69, -21.9, 180.89], [-0.048665, 0.70543, 0.703648, 0.069851], [0,0,0,0], [9E9, 9E9, 9E9, 9E9, 9E9, 9E9]];
	VAR robtarget OpenholeUD_2237 := [[427.69, -21.9, 180.78], [-0.061865, 0.704395, 0.702241, 0.082808], [0,0,0,0], [9E9, 9E9, 9E9, 9E9, 9E9, 9E9]];
	VAR robtarget OpenholeUD_2238 := [[423.7, -21.9, 180.67], [-0.074859, 0.703133, 0.700625, 0.095524], [0,0,0,0], [9E9, 9E9, 9E9, 9E9, 9E9, 9E9]];
	VAR robtarget OpenholeUD_2239 := [[419.7, -21.9, 180.56], [-0.087613, 0.701658, 0.698815, 0.10797], [0,0,0,0], [9E9, 9E9, 9E9, 9E9, 9E9, 9E9]];
	VAR robtarget OpenholeUD_2240 := [[415.7, -21.9, 180.45], [-0.100097, 0.699986, 0.696829, 0.12012], [0,0,0,0], [9E9, 9E9, 9E9, 9E9, 9E9, 9E9]];
	VAR robtarget OpenholeUD_2241 := [[411.7, -21.9, 180.34], [-0.112285, 0.698135, 0.694686, 0.131951], [0,0,0,0], [9E9, 9E9, 9E9, 9E9, 9E9, 9E9]];
	VAR robtarget OpenholeUD_2242 := [[407.7, -21.9, 180.23], [-0.124156, 0.696122, 0.692404, 0.143446], [0,0,0,0], [9E9, 9E9, 9E9, 9E9, 9E9, 9E9]];
	VAR robtarget OpenholeUD_2243 := [[403.7, -21.9, 180.12], [-0.135692, 0.693965, 0.690001, 0.154592], [0,0,0,0], [9E9, 9E9, 9E9, 9E9, 9E9, 9E9]];
	VAR robtarget OpenholeUD_2244 := [[399.7, -21.9, 180.01], [-0.14688, 0.691684, 0.687495, 0.165379], [0,0,0,0], [9E9, 9E9, 9E9, 9E9, 9E9, 9E9]];
	VAR robtarget OpenholeUD_2245 := [[395.71, -21.9, 179.9], [-0.157711, 0.689295, 0.684904, 0.175801], [0,0,0,0], [9E9, 9E9, 9E9, 9E9, 9E9, 9E9]];
	VAR robtarget OpenholeUD_2246 := [[389.34, -21.9, 179.72], [-0.174202, 0.685313, 0.680644, 0.191634], [0,0,0,0], [9E9, 9E9, 9E9, 9E9, 9E9, 9E9]];
	VAR robtarget OpenholeUD_2247 := [[385.34, -21.9, 179.73], [-0.183051, 0.683002, 0.683002, 0.183051], [0,0,0,0], [9E9, 9E9, 9E9, 9E9, 9E9, 9E9]];
	VAR robtarget OpenholeUD_2248 := [[381.34, -21.9, 179.75], [-0.183051, 0.683002, 0.683002, 0.183051], [0,0,0,0], [9E9, 9E9, 9E9, 9E9, 9E9, 9E9]];
	VAR robtarget OpenholeUD_2249 := [[377.34, -21.9, 179.76], [-0.183051, 0.683002, 0.683002, 0.183051], [0,0,0,0], [9E9, 9E9, 9E9, 9E9, 9E9, 9E9]];
	VAR robtarget OpenholeUD_2250 := [[373.34, -21.9, 179.77], [-0.183051, 0.683002, 0.683002, 0.183051], [0,0,0,0], [9E9, 9E9, 9E9, 9E9, 9E9, 9E9]];
	VAR robtarget OpenholeUD_2251 := [[369.34, -21.9, 179.78], [-0.183051, 0.683002, 0.683002, 0.183051], [0,0,0,0], [9E9, 9E9, 9E9, 9E9, 9E9, 9E9]];
	VAR robtarget OpenholeUD_2252 := [[369.34, -21.9, 179.78], [-0.183051, 0.683002, 0.683002, 0.183051], [0,0,0,0], [9E9, 9E9, 9E9, 9E9, 9E9, 9E9]];
	VAR robtarget OpenholeUD_2253 := [[369.34, -23.1, 179.09], [-0.183051, 0.683002, 0.683002, 0.183051], [0,0,0,0], [9E9, 9E9, 9E9, 9E9, 9E9, 9E9]];
	VAR robtarget OpenholeUD_2254 := [[373.34, -23.1, 179.08], [-0.183051, 0.683002, 0.683002, 0.183051], [0,0,0,0], [9E9, 9E9, 9E9, 9E9, 9E9, 9E9]];
	VAR robtarget OpenholeUD_2255 := [[377.34, -23.1, 179.07], [-0.183051, 0.683002, 0.683002, 0.183051], [0,0,0,0], [9E9, 9E9, 9E9, 9E9, 9E9, 9E9]];
	VAR robtarget OpenholeUD_2256 := [[381.34, -23.1, 179.05], [-0.183051, 0.683002, 0.683002, 0.183051], [0,0,0,0], [9E9, 9E9, 9E9, 9E9, 9E9, 9E9]];
	VAR robtarget OpenholeUD_2257 := [[385.34, -23.1, 179.04], [-0.183051, 0.683002, 0.683002, 0.183051], [0,0,0,0], [9E9, 9E9, 9E9, 9E9, 9E9, 9E9]];
	VAR robtarget OpenholeUD_2258 := [[389.34, -23.1, 179.03], [-0.170773, 0.686175, 0.679678, 0.195032], [0,0,0,0], [9E9, 9E9, 9E9, 9E9, 9E9, 9E9]];
	VAR robtarget OpenholeUD_2259 := [[393.34, -23.1, 179.19], [-0.160457, 0.688661, 0.682404, 0.18527], [0,0,0,0], [9E9, 9E9, 9E9, 9E9, 9E9, 9E9]];
	VAR robtarget OpenholeUD_2260 := [[397.33, -23.1, 179.34], [-0.149778, 0.691062, 0.685074, 0.175138], [0,0,0,0], [9E9, 9E9, 9E9, 9E9, 9E9, 9E9]];
	VAR robtarget OpenholeUD_2261 := [[401.33, -23.1, 179.5], [-0.138739, 0.693362, 0.687673, 0.164638], [0,0,0,0], [9E9, 9E9, 9E9, 9E9, 9E9, 9E9]];
	VAR robtarget OpenholeUD_2262 := [[405.33, -23.1, 179.66], [-0.127349, 0.695544, 0.690184, 0.153773], [0,0,0,0], [9E9, 9E9, 9E9, 9E9, 9E9, 9E9]];
	VAR robtarget OpenholeUD_2263 := [[409.32, -23.1, 179.81], [-0.115619, 0.69759, 0.692589, 0.14255], [0,0,0,0], [9E9, 9E9, 9E9, 9E9, 9E9, 9E9]];
	VAR robtarget OpenholeUD_2264 := [[413.32, -23.1, 179.97], [-0.103565, 0.699481, 0.69487, 0.13098], [0,0,0,0], [9E9, 9E9, 9E9, 9E9, 9E9, 9E9]];
	VAR robtarget OpenholeUD_2265 := [[417.32, -23.1, 180.13], [-0.091206, 0.7012, 0.697008, 0.119077], [0,0,0,0], [9E9, 9E9, 9E9, 9E9, 9E9, 9E9]];
	VAR robtarget OpenholeUD_2266 := [[421.31, -23.1, 180.28], [-0.078566, 0.702729, 0.698986, 0.10686], [0,0,0,0], [9E9, 9E9, 9E9, 9E9, 9E9, 9E9]];
	VAR robtarget OpenholeUD_2267 := [[425.31, -23.1, 180.44], [-0.065673, 0.70405, 0.700784, 0.094351], [0,0,0,0], [9E9, 9E9, 9E9, 9E9, 9E9, 9E9]];
	VAR robtarget OpenholeUD_2268 := [[429.31, -23.1, 180.6], [-0.05256, 0.705151, 0.702385, 0.081579], [0,0,0,0], [9E9, 9E9, 9E9, 9E9, 9E9, 9E9]];
	VAR robtarget OpenholeUD_2269 := [[433.3, -23.1, 180.75], [-0.039262, 0.706016, 0.703774, 0.068573], [0,0,0,0], [9E9, 9E9, 9E9, 9E9, 9E9, 9E9]];
	VAR robtarget OpenholeUD_2270 := [[437.3, -23.1, 180.91], [-0.025819, 0.706635, 0.704936, 0.05537], [0,0,0,0], [9E9, 9E9, 9E9, 9E9, 9E9, 9E9]];
	VAR robtarget OpenholeUD_2271 := [[444.56, -23.1, 181.19], [-0.001167, 0.707106, 0.706426, 0.03101], [0,0,0,0], [9E9, 9E9, 9E9, 9E9, 9E9, 9E9]];
	VAR robtarget OpenholeUD_2272 := [[444.56, -23.1, 181.19], [-0.001167, 0.707106, 0.706426, 0.03101], [0,0,0,0], [9E9, 9E9, 9E9, 9E9, 9E9, 9E9]];
	VAR robtarget OpenholeUD_2273 := [[446.05, -24.3, 181.21], [0.007968, 0.707062, 0.706468, 0.030051], [0,0,0,0], [9E9, 9E9, 9E9, 9E9, 9E9, 9E9]];
	VAR robtarget OpenholeUD_2274 := [[442.05, -24.3, 181.01], [-0.005645, 0.707084, 0.705766, 0.043531], [0,0,0,0], [9E9, 9E9, 9E9, 9E9, 9E9, 9E9]];
	VAR robtarget OpenholeUD_2275 := [[438.06, -24.3, 180.81], [-0.019214, 0.706846, 0.704814, 0.056893], [0,0,0,0], [9E9, 9E9, 9E9, 9E9, 9E9, 9E9]];
	VAR robtarget OpenholeUD_2276 := [[434.06, -24.3, 180.61], [-0.032696, 0.70635, 0.703624, 0.070096], [0,0,0,0], [9E9, 9E9, 9E9, 9E9, 9E9, 9E9]];
	VAR robtarget OpenholeUD_2277 := [[430.07, -24.3, 180.4], [-0.046046, 0.705606, 0.702207, 0.083102], [0,0,0,0], [9E9, 9E9, 9E9, 9E9, 9E9, 9E9]];
	VAR robtarget OpenholeUD_2278 := [[426.07, -24.3, 180.2], [-0.059226, 0.704622, 0.700577, 0.095876], [0,0,0,0], [9E9, 9E9, 9E9, 9E9, 9E9, 9E9]];
	VAR robtarget OpenholeUD_2279 := [[422.08, -24.3, 180], [-0.072198, 0.703411, 0.698751, 0.108386], [0,0,0,0], [9E9, 9E9, 9E9, 9E9, 9E9, 9E9]];
	VAR robtarget OpenholeUD_2280 := [[418.08, -24.3, 179.79], [-0.084928, 0.701988, 0.696746, 0.120605], [0,0,0,0], [9E9, 9E9, 9E9, 9E9, 9E9, 9E9]];
	VAR robtarget OpenholeUD_2281 := [[414.09, -24.3, 179.59], [-0.097389, 0.700368, 0.69458, 0.132509], [0,0,0,0], [9E9, 9E9, 9E9, 9E9, 9E9, 9E9]];
	VAR robtarget OpenholeUD_2282 := [[410.09, -24.3, 179.39], [-0.109553, 0.698569, 0.692272, 0.144081], [0,0,0,0], [9E9, 9E9, 9E9, 9E9, 9E9, 9E9]];
	VAR robtarget OpenholeUD_2283 := [[406.1, -24.3, 179.19], [-0.1214, 0.696608, 0.689841, 0.155304], [0,0,0,0], [9E9, 9E9, 9E9, 9E9, 9E9, 9E9]];
	VAR robtarget OpenholeUD_2284 := [[402.1, -24.3, 178.98], [-0.132913, 0.694503, 0.687305, 0.166169], [0,0,0,0], [9E9, 9E9, 9E9, 9E9, 9E9, 9E9]];
	VAR robtarget OpenholeUD_2285 := [[398.11, -24.3, 178.78], [-0.14408, 0.692272, 0.684681, 0.176668], [0,0,0,0], [9E9, 9E9, 9E9, 9E9, 9E9, 9E9]];
	VAR robtarget OpenholeUD_2286 := [[394.11, -24.3, 178.58], [-0.154891, 0.689934, 0.681987, 0.186798], [0,0,0,0], [9E9, 9E9, 9E9, 9E9, 9E9, 9E9]];
	VAR robtarget OpenholeUD_2287 := [[389.34, -24.3, 178.34], [-0.167342, 0.68702, 0.678696, 0.198423], [0,0,0,0], [9E9, 9E9, 9E9, 9E9, 9E9, 9E9]];
	VAR robtarget OpenholeUD_2288 := [[385.34, -24.3, 178.35], [-0.183051, 0.683002, 0.683002, 0.183051], [0,0,0,0], [9E9, 9E9, 9E9, 9E9, 9E9, 9E9]];
	VAR robtarget OpenholeUD_2289 := [[381.34, -24.3, 178.36], [-0.183051, 0.683002, 0.683002, 0.183051], [0,0,0,0], [9E9, 9E9, 9E9, 9E9, 9E9, 9E9]];
	VAR robtarget OpenholeUD_2290 := [[377.34, -24.3, 178.37], [-0.183051, 0.683002, 0.683002, 0.183051], [0,0,0,0], [9E9, 9E9, 9E9, 9E9, 9E9, 9E9]];
	VAR robtarget OpenholeUD_2291 := [[369.34, -24.3, 178.4], [-0.183051, 0.683002, 0.683002, 0.183051], [0,0,0,0], [9E9, 9E9, 9E9, 9E9, 9E9, 9E9]];
	VAR robtarget OpenholeUD_2292 := [[369.34, -24.3, 178.4], [-0.183051, 0.683002, 0.683002, 0.183051], [0,0,0,0], [9E9, 9E9, 9E9, 9E9, 9E9, 9E9]];
	VAR robtarget OpenholeUD_2293 := [[369.33, -25.5, 177.71], [-0.183051, 0.683002, 0.683002, 0.183051], [0,0,0,0], [9E9, 9E9, 9E9, 9E9, 9E9, 9E9]];
	VAR robtarget OpenholeUD_2294 := [[373.33, -25.5, 177.69], [-0.183051, 0.683002, 0.683002, 0.183051], [0,0,0,0], [9E9, 9E9, 9E9, 9E9, 9E9, 9E9]];
	VAR robtarget OpenholeUD_2295 := [[377.33, -25.5, 177.68], [-0.183051, 0.683002, 0.683002, 0.183051], [0,0,0,0], [9E9, 9E9, 9E9, 9E9, 9E9, 9E9]];
	VAR robtarget OpenholeUD_2296 := [[381.33, -25.5, 177.67], [-0.183051, 0.683002, 0.683002, 0.183051], [0,0,0,0], [9E9, 9E9, 9E9, 9E9, 9E9, 9E9]];
	VAR robtarget OpenholeUD_2297 := [[385.33, -25.5, 177.66], [-0.183051, 0.683002, 0.683002, 0.183051], [0,0,0,0], [9E9, 9E9, 9E9, 9E9, 9E9, 9E9]];
	VAR robtarget OpenholeUD_2298 := [[389.33, -25.5, 177.64], [-0.16391, 0.687847, 0.677698, 0.201807], [0,0,0,0], [9E9, 9E9, 9E9, 9E9, 9E9, 9E9]];
	VAR robtarget OpenholeUD_2299 := [[393.33, -25.5, 177.89], [-0.153469, 0.690251, 0.680486, 0.192195], [0,0,0,0], [9E9, 9E9, 9E9, 9E9, 9E9, 9E9]];
	VAR robtarget OpenholeUD_2300 := [[397.32, -25.5, 178.14], [-0.142669, 0.692565, 0.683227, 0.182212], [0,0,0,0], [9E9, 9E9, 9E9, 9E9, 9E9, 9E9]];
	VAR robtarget OpenholeUD_2301 := [[401.31, -25.5, 178.39], [-0.131514, 0.694769, 0.685904, 0.171859], [0,0,0,0], [9E9, 9E9, 9E9, 9E9, 9E9, 9E9]];
	VAR robtarget OpenholeUD_2302 := [[405.3, -25.5, 178.64], [-0.120013, 0.696848, 0.688502, 0.161138], [0,0,0,0], [9E9, 9E9, 9E9, 9E9, 9E9, 9E9]];
	VAR robtarget OpenholeUD_2303 := [[409.3, -25.5, 178.89], [-0.108178, 0.698783, 0.691002, 0.150054], [0,0,0,0], [9E9, 9E9, 9E9, 9E9, 9E9, 9E9]];
	VAR robtarget OpenholeUD_2304 := [[413.29, -25.5, 179.14], [-0.096028, 0.700556, 0.693387, 0.138618], [0,0,0,0], [9E9, 9E9, 9E9, 9E9, 9E9, 9E9]];
	VAR robtarget OpenholeUD_2305 := [[417.28, -25.5, 179.38], [-0.083581, 0.70215, 0.695637, 0.126841], [0,0,0,0], [9E9, 9E9, 9E9, 9E9, 9E9, 9E9]];
	VAR robtarget OpenholeUD_2306 := [[421.27, -25.5, 179.63], [-0.070863, 0.703547, 0.697735, 0.114742], [0,0,0,0], [9E9, 9E9, 9E9, 9E9, 9E9, 9E9]];
	VAR robtarget OpenholeUD_2307 := [[425.26, -25.5, 179.88], [-0.057904, 0.704732, 0.699661, 0.102343], [0,0,0,0], [9E9, 9E9, 9E9, 9E9, 9E9, 9E9]];
	VAR robtarget OpenholeUD_2308 := [[429.26, -25.5, 180.13], [-0.044736, 0.70569, 0.701398, 0.089669], [0,0,0,0], [9E9, 9E9, 9E9, 9E9, 9E9, 9E9]];
	VAR robtarget OpenholeUD_2309 := [[433.25, -25.5, 180.38], [-0.031396, 0.706409, 0.702929, 0.076749], [0,0,0,0], [9E9, 9E9, 9E9, 9E9, 9E9, 9E9]];
	VAR robtarget OpenholeUD_2310 := [[437.24, -25.5, 180.63], [-0.017924, 0.70688, 0.704239, 0.06362], [0,0,0,0], [9E9, 9E9, 9E9, 9E9, 9E9, 9E9]];
	VAR robtarget OpenholeUD_2311 := [[441.23, -25.5, 180.88], [-0.004362, 0.707093, 0.705314, 0.050316], [0,0,0,0], [9E9, 9E9, 9E9, 9E9, 9E9, 9E9]];
	VAR robtarget OpenholeUD_2312 := [[445.23, -25.5, 181.12], [0.009245, 0.707046, 0.706144, 0.036879], [0,0,0,0], [9E9, 9E9, 9E9, 9E9, 9E9, 9E9]];
	VAR robtarget OpenholeUD_2313 := [[449.22, -25.5, 181.37], [0.022853, 0.706737, 0.706721, 0.023352], [0,0,0,0], [9E9, 9E9, 9E9, 9E9, 9E9, 9E9]];
	VAR robtarget OpenholeUD_2314 := [[453.21, -25.5, 181.62], [0.036416, 0.706168, 0.707039, 0.009778], [0,0,0,0], [9E9, 9E9, 9E9, 9E9, 9E9, 9E9]];
	VAR robtarget OpenholeUD_2315 := [[457.2, -25.5, 181.87], [0.049889, 0.705345, 0.707097, -0.003797], [0,0,0,0], [9E9, 9E9, 9E9, 9E9, 9E9, 9E9]];
	VAR robtarget OpenholeUD_2316 := [[461.2, -25.5, 182.12], [0.06323, 0.704274, 0.706894, -0.017329], [0,0,0,0], [9E9, 9E9, 9E9, 9E9, 9E9, 9E9]];
	VAR robtarget OpenholeUD_2317 := [[465.19, -25.5, 182.37], [0.076397, 0.702968, 0.706437, -0.030774], [0,0,0,0], [9E9, 9E9, 9E9, 9E9, 9E9, 9E9]];
	VAR robtarget OpenholeUD_2318 := [[469.18, -25.5, 182.62], [0.089352, 0.701439, 0.705731, -0.04409], [0,0,0,0], [9E9, 9E9, 9E9, 9E9, 9E9, 9E9]];
	VAR robtarget OpenholeUD_2319 := [[473.17, -25.5, 182.87], [0.102062, 0.699702, 0.704786, -0.057237], [0,0,0,0], [9E9, 9E9, 9E9, 9E9, 9E9, 9E9]];
	VAR robtarget OpenholeUD_2320 := [[477.16, -25.5, 183.11], [0.114495, 0.697776, 0.703616, -0.070179], [0,0,0,0], [9E9, 9E9, 9E9, 9E9, 9E9, 9E9]];
	VAR robtarget OpenholeUD_2321 := [[481.16, -25.5, 183.36], [0.126627, 0.695676, 0.702233, -0.082882], [0,0,0,0], [9E9, 9E9, 9E9, 9E9, 9E9, 9E9]];
	VAR robtarget OpenholeUD_2322 := [[485.15, -25.5, 183.61], [0.138434, 0.693424, 0.700653, -0.095319], [0,0,0,0], [9E9, 9E9, 9E9, 9E9, 9E9, 9E9]];
	VAR robtarget OpenholeUD_2323 := [[489.14, -25.5, 183.86], [0.149899, 0.691036, 0.698893, -0.107463], [0,0,0,0], [9E9, 9E9, 9E9, 9E9, 9E9, 9E9]];
	VAR robtarget OpenholeUD_2324 := [[493.13, -25.5, 184.11], [0.161009, 0.688532, 0.696971, -0.119293], [0,0,0,0], [9E9, 9E9, 9E9, 9E9, 9E9, 9E9]];
	VAR robtarget OpenholeUD_2325 := [[497.13, -25.5, 184.36], [0.171754, 0.68593, 0.694905, -0.130794], [0,0,0,0], [9E9, 9E9, 9E9, 9E9, 9E9, 9E9]];
	VAR robtarget OpenholeUD_2326 := [[501.12, -25.5, 184.61], [0.18213, 0.683249, 0.692712, -0.141951], [0,0,0,0], [9E9, 9E9, 9E9, 9E9, 9E9, 9E9]];
	VAR robtarget OpenholeUD_2327 := [[505.11, -25.5, 184.86], [0.192132, 0.680504, 0.69041, -0.152757], [0,0,0,0], [9E9, 9E9, 9E9, 9E9, 9E9, 9E9]];
	VAR robtarget OpenholeUD_2328 := [[509.36, -25.5, 185.12], [0.183051, 0.683002, 0.683002, -0.183051], [0,0,0,0], [9E9, 9E9, 9E9, 9E9, 9E9, 9E9]];
	VAR robtarget OpenholeUD_2329 := [[513.36, -25.5, 185.11], [0.183051, 0.683002, 0.683002, -0.183051], [0,0,0,0], [9E9, 9E9, 9E9, 9E9, 9E9, 9E9]];
	VAR robtarget OpenholeUD_2330 := [[517.36, -25.5, 185.09], [0.183051, 0.683002, 0.683002, -0.183051], [0,0,0,0], [9E9, 9E9, 9E9, 9E9, 9E9, 9E9]];
	VAR robtarget OpenholeUD_2331 := [[521.36, -25.5, 185.08], [0.183051, 0.683002, 0.683002, -0.183051], [0,0,0,0], [9E9, 9E9, 9E9, 9E9, 9E9, 9E9]];
	VAR robtarget OpenholeUD_2332 := [[525.36, -25.5, 185.07], [0.183051, 0.683002, 0.683002, -0.183051], [0,0,0,0], [9E9, 9E9, 9E9, 9E9, 9E9, 9E9]];
	VAR robtarget OpenholeUD_2333 := [[529.36, -25.5, 185.06], [0.183051, 0.683002, 0.683002, -0.183051], [0,0,0,0], [9E9, 9E9, 9E9, 9E9, 9E9, 9E9]];
	VAR robtarget OpenholeUD_2334 := [[529.36, -25.5, 185.06], [0.183051, 0.683002, 0.683002, -0.183051], [0,0,0,0], [9E9, 9E9, 9E9, 9E9, 9E9, 9E9]];
	VAR robtarget OpenholeUD_2335 := [[529.36, -26.7, 185.75], [0.183051, 0.683002, 0.683002, -0.183051], [0,0,0,0], [9E9, 9E9, 9E9, 9E9, 9E9, 9E9]];
	VAR robtarget OpenholeUD_2336 := [[525.36, -26.7, 185.76], [0.183051, 0.683002, 0.683002, -0.183051], [0,0,0,0], [9E9, 9E9, 9E9, 9E9, 9E9, 9E9]];
	VAR robtarget OpenholeUD_2337 := [[521.36, -26.7, 185.78], [0.183051, 0.683002, 0.683002, -0.183051], [0,0,0,0], [9E9, 9E9, 9E9, 9E9, 9E9, 9E9]];
	VAR robtarget OpenholeUD_2338 := [[517.36, -26.7, 185.79], [0.183051, 0.683002, 0.683002, -0.183051], [0,0,0,0], [9E9, 9E9, 9E9, 9E9, 9E9, 9E9]];
	VAR robtarget OpenholeUD_2339 := [[513.36, -26.7, 185.8], [0.183051, 0.683002, 0.683002, -0.183051], [0,0,0,0], [9E9, 9E9, 9E9, 9E9, 9E9, 9E9]];
	VAR robtarget OpenholeUD_2340 := [[509.36, -26.7, 185.81], [0.183051, 0.683002, 0.683002, -0.183051], [0,0,0,0], [9E9, 9E9, 9E9, 9E9, 9E9, 9E9]];
	VAR robtarget OpenholeUD_2341 := [[505.37, -26.7, 185.52], [0.196214, 0.679338, 0.691023, -0.149956], [0,0,0,0], [9E9, 9E9, 9E9, 9E9, 9E9, 9E9]];
	VAR robtarget OpenholeUD_2342 := [[501.38, -26.7, 185.22], [0.186312, 0.68212, 0.693287, -0.139115], [0,0,0,0], [9E9, 9E9, 9E9, 9E9, 9E9, 9E9]];
	VAR robtarget OpenholeUD_2343 := [[497.39, -26.7, 184.93], [0.176037, 0.684844, 0.695439, -0.127925], [0,0,0,0], [9E9, 9E9, 9E9, 9E9, 9E9, 9E9]];
	VAR robtarget OpenholeUD_2344 := [[493.4, -26.7, 184.63], [0.16539, 0.687493, 0.697461, -0.116394], [0,0,0,0], [9E9, 9E9, 9E9, 9E9, 9E9, 9E9]];
	VAR robtarget OpenholeUD_2345 := [[489.41, -26.7, 184.34], [0.154375, 0.690049, 0.699337, -0.104536], [0,0,0,0], [9E9, 9E9, 9E9, 9E9, 9E9, 9E9]];
	VAR robtarget OpenholeUD_2346 := [[485.43, -26.7, 184.05], [0.143003, 0.692496, 0.701048, -0.092367], [0,0,0,0], [9E9, 9E9, 9E9, 9E9, 9E9, 9E9]];
	VAR robtarget OpenholeUD_2347 := [[481.44, -26.7, 183.75], [0.131284, 0.694813, 0.702577, -0.079909], [0,0,0,0], [9E9, 9E9, 9E9, 9E9, 9E9, 9E9]];
	VAR robtarget OpenholeUD_2348 := [[477.45, -26.7, 183.46], [0.119236, 0.696981, 0.703908, -0.067187], [0,0,0,0], [9E9, 9E9, 9E9, 9E9, 9E9, 9E9]];
	VAR robtarget OpenholeUD_2349 := [[473.46, -26.7, 183.16], [0.106879, 0.698983, 0.705024, -0.054229], [0,0,0,0], [9E9, 9E9, 9E9, 9E9, 9E9, 9E9]];
	VAR robtarget OpenholeUD_2350 := [[469.47, -26.7, 182.87], [0.09424, 0.700799, 0.705913, -0.041071], [0,0,0,0], [9E9, 9E9, 9E9, 9E9, 9E9, 9E9]];
	VAR robtarget OpenholeUD_2351 := [[465.48, -26.7, 182.57], [0.081346, 0.702412, 0.706562, -0.027747], [0,0,0,0], [9E9, 9E9, 9E9, 9E9, 9E9, 9E9]];
	VAR robtarget OpenholeUD_2352 := [[461.49, -26.7, 182.28], [0.068233, 0.703807, 0.706962, -0.014298], [0,0,0,0], [9E9, 9E9, 9E9, 9E9, 9E9, 9E9]];
	VAR robtarget OpenholeUD_2353 := [[457.5, -26.7, 181.98], [0.054936, 0.70497, 0.707106, -0.000766], [0,0,0,0], [9E9, 9E9, 9E9, 9E9, 9E9, 9E9]];
	VAR robtarget OpenholeUD_2354 := [[453.51, -26.7, 181.69], [0.041497, 0.705888, 0.706991, 0.012805], [0,0,0,0], [9E9, 9E9, 9E9, 9E9, 9E9, 9E9]];
	VAR robtarget OpenholeUD_2355 := [[449.52, -26.7, 181.39], [0.027957, 0.706554, 0.706615, 0.026371], [0,0,0,0], [9E9, 9E9, 9E9, 9E9, 9E9, 9E9]];
	VAR robtarget OpenholeUD_2356 := [[445.53, -26.7, 181.1], [0.014362, 0.706961, 0.705981, 0.039886], [0,0,0,0], [9E9, 9E9, 9E9, 9E9, 9E9, 9E9]];
	VAR robtarget OpenholeUD_2357 := [[441.55, -26.7, 180.81], [0.000756, 0.707106, 0.705095, 0.053308], [0,0,0,0], [9E9, 9E9, 9E9, 9E9, 9E9, 9E9]];
	VAR robtarget OpenholeUD_2358 := [[437.56, -26.7, 180.51], [-0.012815, 0.706991, 0.703964, 0.066592], [0,0,0,0], [9E9, 9E9, 9E9, 9E9, 9E9, 9E9]];
	VAR robtarget OpenholeUD_2359 := [[433.57, -26.7, 180.22], [-0.026307, 0.706617, 0.702601, 0.079699], [0,0,0,0], [9E9, 9E9, 9E9, 9E9, 9E9, 9E9]];
	VAR robtarget OpenholeUD_2360 := [[429.58, -26.7, 179.92], [-0.039677, 0.705993, 0.701018, 0.092592], [0,0,0,0], [9E9, 9E9, 9E9, 9E9, 9E9, 9E9]];
	VAR robtarget OpenholeUD_2361 := [[425.59, -26.7, 179.63], [-0.052885, 0.705126, 0.699232, 0.105238], [0,0,0,0], [9E9, 9E9, 9E9, 9E9, 9E9, 9E9]];
	VAR robtarget OpenholeUD_2362 := [[421.6, -26.7, 179.33], [-0.065893, 0.70403, 0.697258, 0.117606], [0,0,0,0], [9E9, 9E9, 9E9, 9E9, 9E9, 9E9]];
	VAR robtarget OpenholeUD_2363 := [[417.61, -26.7, 179.04], [-0.078668, 0.702717, 0.695116, 0.12967], [0,0,0,0], [9E9, 9E9, 9E9, 9E9, 9E9, 9E9]];
	VAR robtarget OpenholeUD_2364 := [[413.62, -26.7, 178.74], [-0.091179, 0.701203, 0.692823, 0.14141], [0,0,0,0], [9E9, 9E9, 9E9, 9E9, 9E9, 9E9]];
	VAR robtarget OpenholeUD_2365 := [[409.63, -26.7, 178.45], [-0.103402, 0.699506, 0.690398, 0.152809], [0,0,0,0], [9E9, 9E9, 9E9, 9E9, 9E9, 9E9]];
	VAR robtarget OpenholeUD_2366 := [[405.64, -26.7, 178.15], [-0.115313, 0.697641, 0.687861, 0.163852], [0,0,0,0], [9E9, 9E9, 9E9, 9E9, 9E9, 9E9]];
	VAR robtarget OpenholeUD_2367 := [[401.65, -26.7, 177.86], [-0.126896, 0.695627, 0.685229, 0.174532], [0,0,0,0], [9E9, 9E9, 9E9, 9E9, 9E9, 9E9]];
	VAR robtarget OpenholeUD_2368 := [[397.66, -26.7, 177.57], [-0.138138, 0.693482, 0.68252, 0.184843], [0,0,0,0], [9E9, 9E9, 9E9, 9E9, 9E9, 9E9]];
	VAR robtarget OpenholeUD_2369 := [[393.68, -26.7, 177.27], [-0.149028, 0.691224, 0.67975, 0.194781], [0,0,0,0], [9E9, 9E9, 9E9, 9E9, 9E9, 9E9]];
	VAR robtarget OpenholeUD_2370 := [[389.33, -26.7, 176.95], [-0.160478, 0.688656, 0.676684, 0.205181], [0,0,0,0], [9E9, 9E9, 9E9, 9E9, 9E9, 9E9]];
	VAR robtarget OpenholeUD_2371 := [[385.33, -26.7, 176.96], [-0.183051, 0.683002, 0.683002, 0.183051], [0,0,0,0], [9E9, 9E9, 9E9, 9E9, 9E9, 9E9]];
	VAR robtarget OpenholeUD_2372 := [[381.33, -26.7, 176.98], [-0.183051, 0.683002, 0.683002, 0.183051], [0,0,0,0], [9E9, 9E9, 9E9, 9E9, 9E9, 9E9]];
	VAR robtarget OpenholeUD_2373 := [[377.33, -26.7, 176.99], [-0.183051, 0.683002, 0.683002, 0.183051], [0,0,0,0], [9E9, 9E9, 9E9, 9E9, 9E9, 9E9]];
	VAR robtarget OpenholeUD_2374 := [[373.33, -26.7, 177], [-0.183051, 0.683002, 0.683002, 0.183051], [0,0,0,0], [9E9, 9E9, 9E9, 9E9, 9E9, 9E9]];
	VAR robtarget OpenholeUD_2375 := [[369.33, -26.7, 177.01], [-0.183051, 0.683002, 0.683002, 0.183051], [0,0,0,0], [9E9, 9E9, 9E9, 9E9, 9E9, 9E9]];
	VAR robtarget OpenholeUD_2376 := [[369.33, -26.7, 177.01], [-0.183051, 0.683002, 0.683002, 0.183051], [0,0,0,0], [9E9, 9E9, 9E9, 9E9, 9E9, 9E9]];
	VAR robtarget OpenholeUD_2377 := [[369.33, -27.9, 176.32], [-0.183051, 0.683002, 0.683002, 0.183051], [0,0,0,0], [9E9, 9E9, 9E9, 9E9, 9E9, 9E9]];
	VAR robtarget OpenholeUD_2378 := [[373.33, -27.9, 176.31], [-0.183051, 0.683002, 0.683002, 0.183051], [0,0,0,0], [9E9, 9E9, 9E9, 9E9, 9E9, 9E9]];
	VAR robtarget OpenholeUD_2379 := [[377.33, -27.9, 176.29], [-0.183051, 0.683002, 0.683002, 0.183051], [0,0,0,0], [9E9, 9E9, 9E9, 9E9, 9E9, 9E9]];
	VAR robtarget OpenholeUD_2380 := [[381.33, -27.9, 176.28], [-0.183051, 0.683002, 0.683002, 0.183051], [0,0,0,0], [9E9, 9E9, 9E9, 9E9, 9E9, 9E9]];
	VAR robtarget OpenholeUD_2381 := [[385.33, -27.9, 176.27], [-0.183051, 0.683002, 0.683002, 0.183051], [0,0,0,0], [9E9, 9E9, 9E9, 9E9, 9E9, 9E9]];
	VAR robtarget OpenholeUD_2382 := [[389.33, -27.9, 176.26], [-0.157046, 0.689446, 0.675654, 0.208546], [0,0,0,0], [9E9, 9E9, 9E9, 9E9, 9E9, 9E9]];
	VAR robtarget OpenholeUD_2383 := [[393.32, -27.9, 176.6], [-0.146488, 0.691767, 0.678501, 0.199089], [0,0,0,0], [9E9, 9E9, 9E9, 9E9, 9E9, 9E9]];
	VAR robtarget OpenholeUD_2384 := [[397.3, -27.9, 176.94], [-0.135574, 0.693988, 0.681308, 0.189261], [0,0,0,0], [9E9, 9E9, 9E9, 9E9, 9E9, 9E9]];
	VAR robtarget OpenholeUD_2385 := [[401.29, -27.9, 177.28], [-0.12431, 0.696094, 0.68406, 0.17906], [0,0,0,0], [9E9, 9E9, 9E9, 9E9, 9E9, 9E9]];
	VAR robtarget OpenholeUD_2386 := [[405.27, -27.9, 177.62], [-0.112707, 0.698067, 0.68674, 0.168488], [0,0,0,0], [9E9, 9E9, 9E9, 9E9, 9E9, 9E9]];
	VAR robtarget OpenholeUD_2387 := [[409.26, -27.9, 177.96], [-0.100777, 0.699889, 0.689332, 0.15755], [0,0,0,0], [9E9, 9E9, 9E9, 9E9, 9E9, 9E9]];
	VAR robtarget OpenholeUD_2388 := [[413.24, -27.9, 178.3], [-0.08854, 0.701542, 0.691816, 0.146254], [0,0,0,0], [9E9, 9E9, 9E9, 9E9, 9E9, 9E9]];
	VAR robtarget OpenholeUD_2389 := [[417.23, -27.9, 178.64], [-0.076015, 0.703009, 0.694176, 0.134611], [0,0,0,0], [9E9, 9E9, 9E9, 9E9, 9E9, 9E9]];
	VAR robtarget OpenholeUD_2390 := [[421.21, -27.9, 178.98], [-0.06323, 0.704274, 0.69639, 0.122639], [0,0,0,0], [9E9, 9E9, 9E9, 9E9, 9E9, 9E9]];
	VAR robtarget OpenholeUD_2391 := [[425.2, -27.9, 179.32], [-0.050214, 0.705322, 0.698442, 0.110357], [0,0,0,0], [9E9, 9E9, 9E9, 9E9, 9E9, 9E9]];
	VAR robtarget OpenholeUD_2392 := [[429.19, -27.9, 179.66], [-0.037001, 0.706138, 0.700312, 0.097789], [0,0,0,0], [9E9, 9E9, 9E9, 9E9, 9E9, 9E9]];
	VAR robtarget OpenholeUD_2393 := [[433.17, -27.9, 180], [-0.023629, 0.706712, 0.701983, 0.084966], [0,0,0,0], [9E9, 9E9, 9E9, 9E9, 9E9, 9E9]];
	VAR robtarget OpenholeUD_2394 := [[437.16, -27.9, 180.34], [-0.010138, 0.707034, 0.70344, 0.071919], [0,0,0,0], [9E9, 9E9, 9E9, 9E9, 9E9, 9E9]];
	VAR robtarget OpenholeUD_2395 := [[441.14, -27.9, 180.68], [0.00343, 0.707098, 0.704667, 0.058684], [0,0,0,0], [9E9, 9E9, 9E9, 9E9, 9E9, 9E9]];
	VAR robtarget OpenholeUD_2396 := [[445.13, -27.9, 181.02], [0.017029, 0.706902, 0.705654, 0.045302], [0,0,0,0], [9E9, 9E9, 9E9, 9E9, 9E9, 9E9]];
	VAR robtarget OpenholeUD_2397 := [[449.11, -27.9, 181.36], [0.030616, 0.706444, 0.706391, 0.031814], [0,0,0,0], [9E9, 9E9, 9E9, 9E9, 9E9, 9E9]];
	VAR robtarget OpenholeUD_2398 := [[453.1, -27.9, 181.7], [0.044143, 0.705728, 0.706871, 0.018264], [0,0,0,0], [9E9, 9E9, 9E9, 9E9, 9E9, 9E9]];
	VAR robtarget OpenholeUD_2399 := [[457.08, -27.9, 182.04], [0.057568, 0.704759, 0.707091, 0.004696], [0,0,0,0], [9E9, 9E9, 9E9, 9E9, 9E9, 9E9]];
	VAR robtarget OpenholeUD_2400 := [[461.07, -27.9, 182.38], [0.070848, 0.703549, 0.707051, -0.008844], [0,0,0,0], [9E9, 9E9, 9E9, 9E9, 9E9, 9E9]];
	VAR robtarget OpenholeUD_2401 := [[465.05, -27.9, 182.72], [0.083943, 0.702107, 0.706755, -0.022313], [0,0,0,0], [9E9, 9E9, 9E9, 9E9, 9E9, 9E9]];
	VAR robtarget OpenholeUD_2402 := [[469.04, -27.9, 183.06], [0.096815, 0.700448, 0.706207, -0.035667], [0,0,0,0], [9E9, 9E9, 9E9, 9E9, 9E9, 9E9]];
	VAR robtarget OpenholeUD_2403 := [[473.03, -27.9, 183.4], [0.109431, 0.698588, 0.705416, -0.048868], [0,0,0,0], [9E9, 9E9, 9E9, 9E9, 9E9, 9E9]];
	VAR robtarget OpenholeUD_2404 := [[477.01, -27.9, 183.74], [0.121762, 0.696544, 0.704394, -0.061877], [0,0,0,0], [9E9, 9E9, 9E9, 9E9, 9E9, 9E9]];
	VAR robtarget OpenholeUD_2405 := [[481, -27.9, 184.08], [0.133784, 0.694336, 0.703154, -0.07466], [0,0,0,0], [9E9, 9E9, 9E9, 9E9, 9E9, 9E9]];
	VAR robtarget OpenholeUD_2406 := [[484.98, -27.9, 184.42], [0.145474, 0.691981, 0.701711, -0.087188], [0,0,0,0], [9E9, 9E9, 9E9, 9E9, 9E9, 9E9]];
	VAR robtarget OpenholeUD_2407 := [[488.97, -27.9, 184.76], [0.156817, 0.689499, 0.700081, -0.099434], [0,0,0,0], [9E9, 9E9, 9E9, 9E9, 9E9, 9E9]];
	VAR robtarget OpenholeUD_2408 := [[492.95, -27.9, 185.1], [0.1678, 0.686908, 0.69828, -0.111375], [0,0,0,0], [9E9, 9E9, 9E9, 9E9, 9E9, 9E9]];
	VAR robtarget OpenholeUD_2409 := [[496.94, -27.9, 185.45], [0.178414, 0.684228, 0.696328, -0.122995], [0,0,0,0], [9E9, 9E9, 9E9, 9E9, 9E9, 9E9]];
	VAR robtarget OpenholeUD_2410 := [[500.92, -27.9, 185.79], [0.188656, 0.681475, 0.69424, -0.134278], [0,0,0,0], [9E9, 9E9, 9E9, 9E9, 9E9, 9E9]];
	VAR robtarget OpenholeUD_2411 := [[504.91, -27.9, 186.13], [0.198524, 0.678667, 0.692035, -0.145215], [0,0,0,0], [9E9, 9E9, 9E9, 9E9, 9E9, 9E9]];
	VAR robtarget OpenholeUD_2412 := [[509.36, -27.9, 186.51], [0.183051, 0.683002, 0.683002, -0.183051], [0,0,0,0], [9E9, 9E9, 9E9, 9E9, 9E9, 9E9]];
	VAR robtarget OpenholeUD_2413 := [[513.36, -27.9, 186.49], [0.183051, 0.683002, 0.683002, -0.183051], [0,0,0,0], [9E9, 9E9, 9E9, 9E9, 9E9, 9E9]];
	VAR robtarget OpenholeUD_2414 := [[517.36, -27.9, 186.48], [0.183051, 0.683002, 0.683002, -0.183051], [0,0,0,0], [9E9, 9E9, 9E9, 9E9, 9E9, 9E9]];
	VAR robtarget OpenholeUD_2415 := [[521.36, -27.9, 186.47], [0.183051, 0.683002, 0.683002, -0.183051], [0,0,0,0], [9E9, 9E9, 9E9, 9E9, 9E9, 9E9]];
	VAR robtarget OpenholeUD_2416 := [[525.36, -27.9, 186.46], [0.183051, 0.683002, 0.683002, -0.183051], [0,0,0,0], [9E9, 9E9, 9E9, 9E9, 9E9, 9E9]];
	VAR robtarget OpenholeUD_2417 := [[529.36, -27.9, 186.44], [0.183051, 0.683002, 0.683002, -0.183051], [0,0,0,0], [9E9, 9E9, 9E9, 9E9, 9E9, 9E9]];
	VAR robtarget OpenholeUD_2418 := [[529.36, -27.9, 186.44], [0.183051, 0.683002, 0.683002, -0.183051], [0,0,0,0], [9E9, 9E9, 9E9, 9E9, 9E9, 9E9]];
	VAR robtarget OpenholeUD_2419 := [[529.36, -29.1, 187.14], [0.183051, 0.683002, 0.683002, -0.183051], [0,0,0,0], [9E9, 9E9, 9E9, 9E9, 9E9, 9E9]];
	VAR robtarget OpenholeUD_2420 := [[525.36, -29.1, 187.15], [0.183051, 0.683002, 0.683002, -0.183051], [0,0,0,0], [9E9, 9E9, 9E9, 9E9, 9E9, 9E9]];
	VAR robtarget OpenholeUD_2421 := [[521.36, -29.1, 187.16], [0.183051, 0.683002, 0.683002, -0.183051], [0,0,0,0], [9E9, 9E9, 9E9, 9E9, 9E9, 9E9]];
	VAR robtarget OpenholeUD_2422 := [[517.36, -29.1, 187.17], [0.183051, 0.683002, 0.683002, -0.183051], [0,0,0,0], [9E9, 9E9, 9E9, 9E9, 9E9, 9E9]];
	VAR robtarget OpenholeUD_2423 := [[513.36, -29.1, 187.19], [0.183051, 0.683002, 0.683002, -0.183051], [0,0,0,0], [9E9, 9E9, 9E9, 9E9, 9E9, 9E9]];
	VAR robtarget OpenholeUD_2424 := [[509.36, -29.1, 187.2], [0.183051, 0.683002, 0.683002, -0.183051], [0,0,0,0], [9E9, 9E9, 9E9, 9E9, 9E9, 9E9]];
	VAR robtarget OpenholeUD_2425 := [[505.38, -29.1, 186.81], [0.203092, 0.677314, 0.692496, -0.142999], [0,0,0,0], [9E9, 9E9, 9E9, 9E9, 9E9, 9E9]];
	VAR robtarget OpenholeUD_2426 := [[501.4, -29.1, 186.43], [0.193347, 0.680159, 0.694667, -0.13205], [0,0,0,0], [9E9, 9E9, 9E9, 9E9, 9E9, 9E9]];
	VAR robtarget OpenholeUD_2427 := [[497.42, -29.1, 186.04], [0.183228, 0.682955, 0.696719, -0.120756], [0,0,0,0], [9E9, 9E9, 9E9, 9E9, 9E9, 9E9]];
	VAR robtarget OpenholeUD_2428 := [[493.44, -29.1, 185.66], [0.172734, 0.685684, 0.698635, -0.109128], [0,0,0,0], [9E9, 9E9, 9E9, 9E9, 9E9, 9E9]];
	VAR robtarget OpenholeUD_2429 := [[489.46, -29.1, 185.27], [0.161869, 0.68833, 0.700397, -0.097179], [0,0,0,0], [9E9, 9E9, 9E9, 9E9, 9E9, 9E9]];
	VAR robtarget OpenholeUD_2430 := [[485.48, -29.1, 184.88], [0.150641, 0.690874, 0.701988, -0.084929], [0,0,0,0], [9E9, 9E9, 9E9, 9E9, 9E9, 9E9]];
	VAR robtarget OpenholeUD_2431 := [[481.5, -29.1, 184.5], [0.139061, 0.693298, 0.703391, -0.072398], [0,0,0,0], [9E9, 9E9, 9E9, 9E9, 9E9, 9E9]];
	VAR robtarget OpenholeUD_2432 := [[477.51, -29.1, 184.11], [0.127145, 0.695582, 0.704589, -0.059613], [0,0,0,0], [9E9, 9E9, 9E9, 9E9, 9E9, 9E9]];
	VAR robtarget OpenholeUD_2433 := [[473.53, -29.1, 183.73], [0.114911, 0.697707, 0.705569, -0.046604], [0,0,0,0], [9E9, 9E9, 9E9, 9E9, 9E9, 9E9]];
	VAR robtarget OpenholeUD_2434 := [[469.55, -29.1, 183.34], [0.102384, 0.699655, 0.706317, -0.033405], [0,0,0,0], [9E9, 9E9, 9E9, 9E9, 9E9, 9E9]];
	VAR robtarget OpenholeUD_2435 := [[465.57, -29.1, 182.95], [0.089592, 0.701408, 0.706822, -0.020053], [0,0,0,0], [9E9, 9E9, 9E9, 9E9, 9E9, 9E9]];
	VAR robtarget OpenholeUD_2436 := [[461.59, -29.1, 182.57], [0.076568, 0.702949, 0.707076, -0.00659], [0,0,0,0], [9E9, 9E9, 9E9, 9E9, 9E9, 9E9]];
	VAR robtarget OpenholeUD_2437 := [[457.61, -29.1, 182.18], [0.063347, 0.704264, 0.707073, 0.006944], [0,0,0,0], [9E9, 9E9, 9E9, 9E9, 9E9, 9E9]];
	VAR robtarget OpenholeUD_2438 := [[453.63, -29.1, 181.8], [0.049968, 0.705339, 0.706809, 0.020504], [0,0,0,0], [9E9, 9E9, 9E9, 9E9, 9E9, 9E9]];
	VAR robtarget OpenholeUD_2439 := [[449.64, -29.1, 181.41], [0.036474, 0.706165, 0.706287, 0.034045], [0,0,0,0], [9E9, 9E9, 9E9, 9E9, 9E9, 9E9]];
	VAR robtarget OpenholeUD_2440 := [[445.66, -29.1, 181.02], [0.022909, 0.706736, 0.705508, 0.047523], [0,0,0,0], [9E9, 9E9, 9E9, 9E9, 9E9, 9E9]];
	VAR robtarget OpenholeUD_2441 := [[441.68, -29.1, 180.64], [0.009317, 0.707045, 0.70448, 0.060894], [0,0,0,0], [9E9, 9E9, 9E9, 9E9, 9E9, 9E9]];
	VAR robtarget OpenholeUD_2442 := [[437.7, -29.1, 180.25], [-0.004257, 0.707094, 0.703212, 0.074116], [0,0,0,0], [9E9, 9E9, 9E9, 9E9, 9E9, 9E9]];
	VAR robtarget OpenholeUD_2443 := [[433.72, -29.1, 179.87], [-0.017768, 0.706884, 0.701716, 0.08715], [0,0,0,0], [9E9, 9E9, 9E9, 9E9, 9E9, 9E9]];
	VAR robtarget OpenholeUD_2444 := [[429.74, -29.1, 179.48], [-0.031172, 0.706419, 0.700006, 0.099959], [0,0,0,0], [9E9, 9E9, 9E9, 9E9, 9E9, 9E9]];
	VAR robtarget OpenholeUD_2445 := [[425.76, -29.1, 179.09], [-0.044429, 0.70571, 0.698098, 0.112511], [0,0,0,0], [9E9, 9E9, 9E9, 9E9, 9E9, 9E9]];
	VAR robtarget OpenholeUD_2446 := [[421.78, -29.1, 178.71], [-0.0575, 0.704765, 0.696011, 0.124776], [0,0,0,0], [9E9, 9E9, 9E9, 9E9, 9E9, 9E9]];
	VAR robtarget OpenholeUD_2447 := [[417.79, -29.1, 178.32], [-0.070351, 0.703598, 0.693761, 0.136731], [0,0,0,0], [9E9, 9E9, 9E9, 9E9, 9E9, 9E9]];
	VAR robtarget OpenholeUD_2448 := [[413.81, -29.1, 177.94], [-0.082951, 0.702224, 0.691369, 0.148355], [0,0,0,0], [9E9, 9E9, 9E9, 9E9, 9E9, 9E9]];
	VAR robtarget OpenholeUD_2449 := [[409.83, -29.1, 177.55], [-0.095273, 0.700659, 0.688852, 0.159632], [0,0,0,0], [9E9, 9E9, 9E9, 9E9, 9E9, 9E9]];
	VAR robtarget OpenholeUD_2450 := [[405.85, -29.1, 177.17], [-0.107293, 0.698919, 0.686231, 0.17055], [0,0,0,0], [9E9, 9E9, 9E9, 9E9, 9E9, 9E9]];
	VAR robtarget OpenholeUD_2451 := [[401.87, -29.1, 176.78], [-0.118993, 0.697023, 0.683522, 0.181101], [0,0,0,0], [9E9, 9E9, 9E9, 9E9, 9E9, 9E9]];
	VAR robtarget OpenholeUD_2452 := [[397.89, -29.1, 176.39], [-0.130359, 0.694987, 0.680744, 0.191279], [0,0,0,0], [9E9, 9E9, 9E9, 9E9, 9E9, 9E9]];
	VAR robtarget OpenholeUD_2453 := [[393.91, -29.1, 176.01], [-0.14138, 0.692829, 0.677912, 0.201085], [0,0,0,0], [9E9, 9E9, 9E9, 9E9, 9E9, 9E9]];
	VAR robtarget OpenholeUD_2454 := [[389.33, -29.1, 175.56], [-0.153616, 0.690219, 0.67461, 0.211901], [0,0,0,0], [9E9, 9E9, 9E9, 9E9, 9E9, 9E9]];
	VAR robtarget OpenholeUD_2455 := [[385.33, -29.1, 175.58], [-0.183051, 0.683002, 0.683002, 0.183051], [0,0,0,0], [9E9, 9E9, 9E9, 9E9, 9E9, 9E9]];
	VAR robtarget OpenholeUD_2456 := [[381.33, -29.1, 175.59], [-0.183051, 0.683002, 0.683002, 0.183051], [0,0,0,0], [9E9, 9E9, 9E9, 9E9, 9E9, 9E9]];
	VAR robtarget OpenholeUD_2457 := [[377.33, -29.1, 175.6], [-0.183051, 0.683002, 0.683002, 0.183051], [0,0,0,0], [9E9, 9E9, 9E9, 9E9, 9E9, 9E9]];
	VAR robtarget OpenholeUD_2458 := [[373.33, -29.1, 175.61], [-0.183051, 0.683002, 0.683002, 0.183051], [0,0,0,0], [9E9, 9E9, 9E9, 9E9, 9E9, 9E9]];
	VAR robtarget OpenholeUD_2459 := [[369.33, -29.1, 175.63], [-0.183051, 0.683002, 0.683002, 0.183051], [0,0,0,0], [9E9, 9E9, 9E9, 9E9, 9E9, 9E9]];
	VAR robtarget OpenholeUD_2460 := [[369.33, -29.1, 175.63], [-0.183051, 0.683002, 0.683002, 0.183051], [0,0,0,0], [9E9, 9E9, 9E9, 9E9, 9E9, 9E9]];
	VAR robtarget OpenholeUD_2461 := [[369.33, -30.3, 174.93], [-0.183051, 0.683002, 0.683002, 0.183051], [0,0,0,0], [9E9, 9E9, 9E9, 9E9, 9E9, 9E9]];
	VAR robtarget OpenholeUD_2462 := [[373.33, -30.3, 174.92], [-0.183051, 0.683002, 0.683002, 0.183051], [0,0,0,0], [9E9, 9E9, 9E9, 9E9, 9E9, 9E9]];
	VAR robtarget OpenholeUD_2463 := [[377.33, -30.3, 174.91], [-0.183051, 0.683002, 0.683002, 0.183051], [0,0,0,0], [9E9, 9E9, 9E9, 9E9, 9E9, 9E9]];
	VAR robtarget OpenholeUD_2464 := [[381.33, -30.3, 174.9], [-0.183051, 0.683002, 0.683002, 0.183051], [0,0,0,0], [9E9, 9E9, 9E9, 9E9, 9E9, 9E9]];
	VAR robtarget OpenholeUD_2465 := [[385.33, -30.3, 174.88], [-0.183051, 0.683002, 0.683002, 0.183051], [0,0,0,0], [9E9, 9E9, 9E9, 9E9, 9E9, 9E9]];
	VAR robtarget OpenholeUD_2466 := [[389.33, -30.3, 174.87], [-0.150187, 0.690973, 0.67355, 0.215245], [0,0,0,0], [9E9, 9E9, 9E9, 9E9, 9E9, 9E9]];
	VAR robtarget OpenholeUD_2467 := [[393.3, -30.3, 175.3], [-0.139519, 0.693206, 0.676451, 0.205946], [0,0,0,0], [9E9, 9E9, 9E9, 9E9, 9E9, 9E9]];
	VAR robtarget OpenholeUD_2468 := [[397.28, -30.3, 175.73], [-0.1285, 0.695333, 0.67932, 0.196276], [0,0,0,0], [9E9, 9E9, 9E9, 9E9, 9E9, 9E9]];
	VAR robtarget OpenholeUD_2469 := [[401.26, -30.3, 176.17], [-0.117136, 0.697337, 0.682142, 0.186233], [0,0,0,0], [9E9, 9E9, 9E9, 9E9, 9E9, 9E9]];
	VAR robtarget OpenholeUD_2470 := [[405.23, -30.3, 176.6], [-0.10544, 0.699201, 0.684901, 0.175816], [0,0,0,0], [9E9, 9E9, 9E9, 9E9, 9E9, 9E9]];
	VAR robtarget OpenholeUD_2471 := [[409.21, -30.3, 177.03], [-0.093425, 0.700908, 0.687579, 0.165029], [0,0,0,0], [9E9, 9E9, 9E9, 9E9, 9E9, 9E9]];
	VAR robtarget OpenholeUD_2472 := [[413.19, -30.3, 177.46], [-0.081109, 0.70244, 0.69016, 0.153879], [0,0,0,0], [9E9, 9E9, 9E9, 9E9, 9E9, 9E9]];
	VAR robtarget OpenholeUD_2473 := [[417.16, -30.3, 177.89], [-0.068517, 0.703779, 0.692624, 0.142378], [0,0,0,0], [9E9, 9E9, 9E9, 9E9, 9E9, 9E9]];
	VAR robtarget OpenholeUD_2474 := [[421.14, -30.3, 178.32], [-0.055674, 0.704912, 0.694953, 0.130539], [0,0,0,0], [9E9, 9E9, 9E9, 9E9, 9E9, 9E9]];
	VAR robtarget OpenholeUD_2475 := [[425.12, -30.3, 178.75], [-0.042611, 0.705822, 0.697127, 0.118382], [0,0,0,0], [9E9, 9E9, 9E9, 9E9, 9E9, 9E9]];
	VAR robtarget OpenholeUD_2476 := [[429.09, -30.3, 179.18], [-0.029364, 0.706497, 0.699127, 0.10593], [0,0,0,0], [9E9, 9E9, 9E9, 9E9, 9E9, 9E9]];
	VAR robtarget OpenholeUD_2477 := [[433.07, -30.3, 179.62], [-0.015969, 0.706926, 0.700936, 0.093211], [0,0,0,0], [9E9, 9E9, 9E9, 9E9, 9E9, 9E9]];
	VAR robtarget OpenholeUD_2478 := [[437.05, -30.3, 180.05], [-0.002468, 0.707102, 0.702538, 0.080256], [0,0,0,0], [9E9, 9E9, 9E9, 9E9, 9E9, 9E9]];
	VAR robtarget OpenholeUD_2479 := [[441.02, -30.3, 180.48], [0.011096, 0.70702, 0.703916, 0.0671], [0,0,0,0], [9E9, 9E9, 9E9, 9E9, 9E9, 9E9]];
	VAR robtarget OpenholeUD_2480 := [[445, -30.3, 180.91], [0.024679, 0.706676, 0.705058, 0.053782], [0,0,0,0], [9E9, 9E9, 9E9, 9E9, 9E9, 9E9]];
	VAR robtarget OpenholeUD_2481 := [[448.98, -30.3, 181.34], [0.038236, 0.706072, 0.705955, 0.040344], [0,0,0,0], [9E9, 9E9, 9E9, 9E9, 9E9, 9E9]];
	VAR robtarget OpenholeUD_2482 := [[452.95, -30.3, 181.77], [0.051721, 0.705213, 0.706598, 0.026827], [0,0,0,0], [9E9, 9E9, 9E9, 9E9, 9E9, 9E9]];
	VAR robtarget OpenholeUD_2483 := [[456.93, -30.3, 182.2], [0.065092, 0.704104, 0.706982, 0.013277], [0,0,0,0], [9E9, 9E9, 9E9, 9E9, 9E9, 9E9]];
	VAR robtarget OpenholeUD_2484 := [[460.91, -30.3, 182.64], [0.078305, 0.702758, 0.707107, -0.000261], [0,0,0,0], [9E9, 9E9, 9E9, 9E9, 9E9, 9E9]];
	VAR robtarget OpenholeUD_2485 := [[464.88, -30.3, 183.07], [0.091323, 0.701185, 0.706973, -0.013744], [0,0,0,0], [9E9, 9E9, 9E9, 9E9, 9E9, 9E9]];
	VAR robtarget OpenholeUD_2486 := [[468.86, -30.3, 183.5], [0.104107, 0.699401, 0.706586, -0.027129], [0,0,0,0], [9E9, 9E9, 9E9, 9E9, 9E9, 9E9]];
	VAR robtarget OpenholeUD_2487 := [[472.84, -30.3, 183.93], [0.116627, 0.697422, 0.705953, -0.040374], [0,0,0,0], [9E9, 9E9, 9E9, 9E9, 9E9, 9E9]];
	VAR robtarget OpenholeUD_2488 := [[476.81, -30.3, 184.36], [0.128854, 0.695267, 0.705084, -0.053442], [0,0,0,0], [9E9, 9E9, 9E9, 9E9, 9E9, 9E9]];
	VAR robtarget OpenholeUD_2489 := [[480.79, -30.3, 184.79], [0.140764, 0.692954, 0.703992, -0.066298], [0,0,0,0], [9E9, 9E9, 9E9, 9E9, 9E9, 9E9]];
	VAR robtarget OpenholeUD_2490 := [[484.77, -30.3, 185.22], [0.152336, 0.690502, 0.70269, -0.07891], [0,0,0,0], [9E9, 9E9, 9E9, 9E9, 9E9, 9E9]];
	VAR robtarget OpenholeUD_2491 := [[488.74, -30.3, 185.65], [0.163557, 0.687931, 0.701194, -0.091252], [0,0,0,0], [9E9, 9E9, 9E9, 9E9, 9E9, 9E9]];
	VAR robtarget OpenholeUD_2492 := [[492.72, -30.3, 186.09], [0.174413, 0.685259, 0.699521, -0.103299], [0,0,0,0], [9E9, 9E9, 9E9, 9E9, 9E9, 9E9]];
	VAR robtarget OpenholeUD_2493 := [[496.7, -30.3, 186.52], [0.184898, 0.682505, 0.697687, -0.115033], [0,0,0,0], [9E9, 9E9, 9E9, 9E9, 9E9, 9E9]];
	VAR robtarget OpenholeUD_2494 := [[500.67, -30.3, 186.95], [0.195008, 0.679685, 0.695711, -0.126437], [0,0,0,0], [9E9, 9E9, 9E9, 9E9, 9E9, 9E9]];
	VAR robtarget OpenholeUD_2495 := [[504.65, -30.3, 187.38], [0.204743, 0.676816, 0.693609, -0.137502], [0,0,0,0], [9E9, 9E9, 9E9, 9E9, 9E9, 9E9]];
	VAR robtarget OpenholeUD_2496 := [[509.37, -30.3, 187.89], [0.183051, 0.683002, 0.683002, -0.183051], [0,0,0,0], [9E9, 9E9, 9E9, 9E9, 9E9, 9E9]];
	VAR robtarget OpenholeUD_2497 := [[513.37, -30.3, 187.88], [0.183051, 0.683002, 0.683002, -0.183051], [0,0,0,0], [9E9, 9E9, 9E9, 9E9, 9E9, 9E9]];
	VAR robtarget OpenholeUD_2498 := [[517.37, -30.3, 187.87], [0.183051, 0.683002, 0.683002, -0.183051], [0,0,0,0], [9E9, 9E9, 9E9, 9E9, 9E9, 9E9]];
	VAR robtarget OpenholeUD_2499 := [[521.37, -30.3, 187.85], [0.183051, 0.683002, 0.683002, -0.183051], [0,0,0,0], [9E9, 9E9, 9E9, 9E9, 9E9, 9E9]];
	VAR robtarget OpenholeUD_2500 := [[525.37, -30.3, 187.84], [0.183051, 0.683002, 0.683002, -0.183051], [0,0,0,0], [9E9, 9E9, 9E9, 9E9, 9E9, 9E9]];
	VAR robtarget OpenholeUD_2501 := [[529.37, -30.3, 187.83], [0.183051, 0.683002, 0.683002, -0.183051], [0,0,0,0], [9E9, 9E9, 9E9, 9E9, 9E9, 9E9]];
	VAR robtarget OpenholeUD_2502 := [[529.37, -30.3, 187.83], [0.183051, 0.683002, 0.683002, -0.183051], [0,0,0,0], [9E9, 9E9, 9E9, 9E9, 9E9, 9E9]];
	VAR robtarget OpenholeUD_2503 := [[529.37, -31.5, 188.52], [0.183051, 0.683002, 0.683002, -0.183051], [0,0,0,0], [9E9, 9E9, 9E9, 9E9, 9E9, 9E9]];
	VAR robtarget OpenholeUD_2504 := [[525.37, -31.5, 188.53], [0.183051, 0.683002, 0.683002, -0.183051], [0,0,0,0], [9E9, 9E9, 9E9, 9E9, 9E9, 9E9]];
	VAR robtarget OpenholeUD_2505 := [[521.37, -31.5, 188.55], [0.183051, 0.683002, 0.683002, -0.183051], [0,0,0,0], [9E9, 9E9, 9E9, 9E9, 9E9, 9E9]];
	VAR robtarget OpenholeUD_2506 := [[517.37, -31.5, 188.56], [0.183051, 0.683002, 0.683002, -0.183051], [0,0,0,0], [9E9, 9E9, 9E9, 9E9, 9E9, 9E9]];
	VAR robtarget OpenholeUD_2507 := [[513.37, -31.5, 188.57], [0.183051, 0.683002, 0.683002, -0.183051], [0,0,0,0], [9E9, 9E9, 9E9, 9E9, 9E9, 9E9]];
	VAR robtarget OpenholeUD_2508 := [[509.37, -31.5, 188.58], [0.183051, 0.683002, 0.683002, -0.183051], [0,0,0,0], [9E9, 9E9, 9E9, 9E9, 9E9, 9E9]];
	VAR robtarget OpenholeUD_2509 := [[505.4, -31.5, 188.11], [0.209928, 0.675226, 0.693893, -0.136059], [0,0,0,0], [9E9, 9E9, 9E9, 9E9, 9E9, 9E9]];
	VAR robtarget OpenholeUD_2510 := [[501.43, -31.5, 187.63], [0.200345, 0.678131, 0.695969, -0.125009], [0,0,0,0], [9E9, 9E9, 9E9, 9E9, 9E9, 9E9]];
	VAR robtarget OpenholeUD_2511 := [[497.45, -31.5, 187.16], [0.190386, 0.680994, 0.697919, -0.113621], [0,0,0,0], [9E9, 9E9, 9E9, 9E9, 9E9, 9E9]];
	VAR robtarget OpenholeUD_2512 := [[493.48, -31.5, 186.68], [0.18005, 0.6838, 0.699725, -0.101904], [0,0,0,0], [9E9, 9E9, 9E9, 9E9, 9E9, 9E9]];
	VAR robtarget OpenholeUD_2513 := [[489.51, -31.5, 186.2], [0.16934, 0.68653, 0.701372, -0.089875], [0,0,0,0], [9E9, 9E9, 9E9, 9E9, 9E9, 9E9]];
	VAR robtarget OpenholeUD_2514 := [[485.54, -31.5, 185.73], [0.158263, 0.689168, 0.702841, -0.077552], [0,0,0,0], [9E9, 9E9, 9E9, 9E9, 9E9, 9E9]];
	VAR robtarget OpenholeUD_2515 := [[481.57, -31.5, 185.25], [0.146829, 0.691694, 0.704117, -0.064958], [0,0,0,0], [9E9, 9E9, 9E9, 9E9, 9E9, 9E9]];
	VAR robtarget OpenholeUD_2516 := [[477.6, -31.5, 184.77], [0.135051, 0.69409, 0.705183, -0.05212], [0,0,0,0], [9E9, 9E9, 9E9, 9E9, 9E9, 9E9]];
	VAR robtarget OpenholeUD_2517 := [[473.63, -31.5, 184.3], [0.122948, 0.696336, 0.706027, -0.03907], [0,0,0,0], [9E9, 9E9, 9E9, 9E9, 9E9, 9E9]];
	VAR robtarget OpenholeUD_2518 := [[469.65, -31.5, 183.82], [0.110542, 0.698413, 0.706634, -0.025841], [0,0,0,0], [9E9, 9E9, 9E9, 9E9, 9E9, 9E9]];
	VAR robtarget OpenholeUD_2519 := [[465.68, -31.5, 183.34], [0.097861, 0.700302, 0.706997, -0.012471], [0,0,0,0], [9E9, 9E9, 9E9, 9E9, 9E9, 9E9]];
	VAR robtarget OpenholeUD_2520 := [[461.71, -31.5, 182.87], [0.084934, 0.701987, 0.707106, 0.000999], [0,0,0,0], [9E9, 9E9, 9E9, 9E9, 9E9, 9E9]];
	VAR robtarget OpenholeUD_2521 := [[457.74, -31.5, 182.39], [0.071798, 0.703452, 0.706958, 0.014526], [0,0,0,0], [9E9, 9E9, 9E9, 9E9, 9E9, 9E9]];
	VAR robtarget OpenholeUD_2522 := [[453.77, -31.5, 181.91], [0.058491, 0.704684, 0.70655, 0.028066], [0,0,0,0], [9E9, 9E9, 9E9, 9E9, 9E9, 9E9]];
	VAR robtarget OpenholeUD_2523 := [[449.8, -31.5, 181.44], [0.045052, 0.70567, 0.705884, 0.041575], [0,0,0,0], [9E9, 9E9, 9E9, 9E9, 9E9, 9E9]];
	VAR robtarget OpenholeUD_2524 := [[445.83, -31.5, 180.96], [0.031527, 0.706404, 0.704964, 0.055008], [0,0,0,0], [9E9, 9E9, 9E9, 9E9, 9E9, 9E9]];
	VAR robtarget OpenholeUD_2525 := [[441.85, -31.5, 180.48], [0.017959, 0.706879, 0.703798, 0.068323], [0,0,0,0], [9E9, 9E9, 9E9, 9E9, 9E9, 9E9]];
	VAR robtarget OpenholeUD_2526 := [[437.88, -31.5, 180.01], [0.004392, 0.707093, 0.702397, 0.081478], [0,0,0,0], [9E9, 9E9, 9E9, 9E9, 9E9, 9E9]];
	VAR robtarget OpenholeUD_2527 := [[433.91, -31.5, 179.53], [-0.009127, 0.707048, 0.700773, 0.094433], [0,0,0,0], [9E9, 9E9, 9E9, 9E9, 9E9, 9E9]];
	VAR robtarget OpenholeUD_2528 := [[429.94, -31.5, 179.05], [-0.022555, 0.706747, 0.698941, 0.107155], [0,0,0,0], [9E9, 9E9, 9E9, 9E9, 9E9, 9E9]];
	VAR robtarget OpenholeUD_2529 := [[425.97, -31.5, 178.58], [-0.035852, 0.706197, 0.696917, 0.11961], [0,0,0,0], [9E9, 9E9, 9E9, 9E9, 9E9, 9E9]];
	VAR robtarget OpenholeUD_2530 := [[422, -31.5, 178.1], [-0.048978, 0.705408, 0.69472, 0.131772], [0,0,0,0], [9E9, 9E9, 9E9, 9E9, 9E9, 9E9]];
	VAR robtarget OpenholeUD_2531 := [[418.02, -31.5, 177.62], [-0.061898, 0.704392, 0.692369, 0.143616], [0,0,0,0], [9E9, 9E9, 9E9, 9E9, 9E9, 9E9]];
	VAR robtarget OpenholeUD_2532 := [[414.05, -31.5, 177.15], [-0.074578, 0.703163, 0.689882, 0.155123], [0,0,0,0], [9E9, 9E9, 9E9, 9E9, 9E9, 9E9]];
	VAR robtarget OpenholeUD_2533 := [[410.08, -31.5, 176.67], [-0.086993, 0.701735, 0.687278, 0.166279], [0,0,0,0], [9E9, 9E9, 9E9, 9E9, 9E9, 9E9]];
	VAR robtarget OpenholeUD_2534 := [[406.11, -31.5, 176.19], [-0.099116, 0.700126, 0.684577, 0.177071], [0,0,0,0], [9E9, 9E9, 9E9, 9E9, 9E9, 9E9]];
	VAR robtarget OpenholeUD_2535 := [[402.14, -31.5, 175.72], [-0.110929, 0.698352, 0.681796, 0.187494], [0,0,0,0], [9E9, 9E9, 9E9, 9E9, 9E9, 9E9]];
	VAR robtarget OpenholeUD_2536 := [[398.17, -31.5, 175.24], [-0.122415, 0.69643, 0.678953, 0.197543], [0,0,0,0], [9E9, 9E9, 9E9, 9E9, 9E9, 9E9]];
	VAR robtarget OpenholeUD_2537 := [[394.2, -31.5, 174.76], [-0.133562, 0.694378, 0.676063, 0.207217], [0,0,0,0], [9E9, 9E9, 9E9, 9E9, 9E9, 9E9]];
	VAR robtarget OpenholeUD_2538 := [[389.32, -31.5, 174.18], [-0.146762, 0.691709, 0.672476, 0.218577], [0,0,0,0], [9E9, 9E9, 9E9, 9E9, 9E9, 9E9]];
	VAR robtarget OpenholeUD_2539 := [[385.32, -31.5, 174.19], [-0.183051, 0.683002, 0.683002, 0.183051], [0,0,0,0], [9E9, 9E9, 9E9, 9E9, 9E9, 9E9]];
	VAR robtarget OpenholeUD_2540 := [[381.32, -31.5, 174.2], [-0.183051, 0.683002, 0.683002, 0.183051], [0,0,0,0], [9E9, 9E9, 9E9, 9E9, 9E9, 9E9]];
	VAR robtarget OpenholeUD_2541 := [[377.32, -31.5, 174.22], [-0.183051, 0.683002, 0.683002, 0.183051], [0,0,0,0], [9E9, 9E9, 9E9, 9E9, 9E9, 9E9]];
	VAR robtarget OpenholeUD_2542 := [[373.32, -31.5, 174.23], [-0.183051, 0.683002, 0.683002, 0.183051], [0,0,0,0], [9E9, 9E9, 9E9, 9E9, 9E9, 9E9]];
	VAR robtarget OpenholeUD_2543 := [[369.32, -31.5, 174.24], [-0.183051, 0.683002, 0.683002, 0.183051], [0,0,0,0], [9E9, 9E9, 9E9, 9E9, 9E9, 9E9]];
	VAR robtarget OpenholeUD_2544 := [[369.32, -31.5, 174.24], [-0.183051, 0.683002, 0.683002, 0.183051], [0,0,0,0], [9E9, 9E9, 9E9, 9E9, 9E9, 9E9]];
	VAR robtarget OpenholeUD_2545 := [[369.32, -32.7, 173.55], [-0.183051, 0.683002, 0.683002, 0.183051], [0,0,0,0], [9E9, 9E9, 9E9, 9E9, 9E9, 9E9]];
	VAR robtarget OpenholeUD_2546 := [[373.32, -32.7, 173.54], [-0.183051, 0.683002, 0.683002, 0.183051], [0,0,0,0], [9E9, 9E9, 9E9, 9E9, 9E9, 9E9]];
	VAR robtarget OpenholeUD_2547 := [[377.32, -32.7, 173.52], [-0.183051, 0.683002, 0.683002, 0.183051], [0,0,0,0], [9E9, 9E9, 9E9, 9E9, 9E9, 9E9]];
	VAR robtarget OpenholeUD_2548 := [[381.32, -32.7, 173.51], [-0.183051, 0.683002, 0.683002, 0.183051], [0,0,0,0], [9E9, 9E9, 9E9, 9E9, 9E9, 9E9]];
	VAR robtarget OpenholeUD_2549 := [[385.32, -32.7, 173.5], [-0.183051, 0.683002, 0.683002, 0.183051], [0,0,0,0], [9E9, 9E9, 9E9, 9E9, 9E9, 9E9]];
	VAR robtarget OpenholeUD_2550 := [[389.32, -32.7, 173.48], [-0.14334, 0.692426, 0.671388, 0.221897], [0,0,0,0], [9E9, 9E9, 9E9, 9E9, 9E9, 9E9]];
	VAR robtarget OpenholeUD_2551 := [[393.29, -32.7, 174.01], [-0.13257, 0.694568, 0.674339, 0.21276], [0,0,0,0], [9E9, 9E9, 9E9, 9E9, 9E9, 9E9]];
	VAR robtarget OpenholeUD_2552 := [[397.25, -32.7, 174.53], [-0.121454, 0.696598, 0.677265, 0.203252], [0,0,0,0], [9E9, 9E9, 9E9, 9E9, 9E9, 9E9]];
	VAR robtarget OpenholeUD_2553 := [[401.22, -32.7, 175.05], [-0.11, 0.698498, 0.680153, 0.19337], [0,0,0,0], [9E9, 9E9, 9E9, 9E9, 9E9, 9E9]];
	VAR robtarget OpenholeUD_2554 := [[405.18, -32.7, 175.57], [-0.098219, 0.700252, 0.682986, 0.183112], [0,0,0,0], [9E9, 9E9, 9E9, 9E9, 9E9, 9E9]];
	VAR robtarget OpenholeUD_2555 := [[409.15, -32.7, 176.09], [-0.086128, 0.701842, 0.685748, 0.172481], [0,0,0,0], [9E9, 9E9, 9E9, 9E9, 9E9, 9E9]];
	VAR robtarget OpenholeUD_2556 := [[413.12, -32.7, 176.62], [-0.073745, 0.703251, 0.688421, 0.161484], [0,0,0,0], [9E9, 9E9, 9E9, 9E9, 9E9, 9E9]];
	VAR robtarget OpenholeUD_2557 := [[417.08, -32.7, 177.14], [-0.061095, 0.704463, 0.690986, 0.15013], [0,0,0,0], [9E9, 9E9, 9E9, 9E9, 9E9, 9E9]];
	VAR robtarget OpenholeUD_2558 := [[421.05, -32.7, 177.66], [-0.048204, 0.705462, 0.693424, 0.138432], [0,0,0,0], [9E9, 9E9, 9E9, 9E9, 9E9, 9E9]];
	VAR robtarget OpenholeUD_2559 := [[425.01, -32.7, 178.18], [-0.035105, 0.706235, 0.695716, 0.126408], [0,0,0,0], [9E9, 9E9, 9E9, 9E9, 9E9, 9E9]];
	VAR robtarget OpenholeUD_2560 := [[428.98, -32.7, 178.7], [-0.021832, 0.70677, 0.697844, 0.114079], [0,0,0,0], [9E9, 9E9, 9E9, 9E9, 9E9, 9E9]];
	VAR robtarget OpenholeUD_2561 := [[432.95, -32.7, 179.22], [-0.008425, 0.707057, 0.699788, 0.101473], [0,0,0,0], [9E9, 9E9, 9E9, 9E9, 9E9, 9E9]];
	VAR robtarget OpenholeUD_2562 := [[436.91, -32.7, 179.75], [0.005077, 0.707089, 0.701532, 0.088619], [0,0,0,0], [9E9, 9E9, 9E9, 9E9, 9E9, 9E9]];
	VAR robtarget OpenholeUD_2563 := [[440.88, -32.7, 180.27], [0.018629, 0.706861, 0.703059, 0.075552], [0,0,0,0], [9E9, 9E9, 9E9, 9E9, 9E9, 9E9]];
	VAR robtarget OpenholeUD_2564 := [[444.84, -32.7, 180.79], [0.032188, 0.706374, 0.704356, 0.062308], [0,0,0,0], [9E9, 9E9, 9E9, 9E9, 9E9, 9E9]];
	VAR robtarget OpenholeUD_2565 := [[448.81, -32.7, 181.31], [0.045707, 0.705628, 0.705412, 0.048929], [0,0,0,0], [9E9, 9E9, 9E9, 9E9, 9E9, 9E9]];
	VAR robtarget OpenholeUD_2566 := [[452.77, -32.7, 181.83], [0.059144, 0.704629, 0.706217, 0.035457], [0,0,0,0], [9E9, 9E9, 9E9, 9E9, 9E9, 9E9]];
	VAR robtarget OpenholeUD_2567 := [[456.74, -32.7, 182.35], [0.072454, 0.703385, 0.706766, 0.021935], [0,0,0,0], [9E9, 9E9, 9E9, 9E9, 9E9, 9E9]];
	VAR robtarget OpenholeUD_2568 := [[460.71, -32.7, 182.88], [0.085596, 0.701907, 0.707057, 0.008408], [0,0,0,0], [9E9, 9E9, 9E9, 9E9, 9E9, 9E9]];
	VAR robtarget OpenholeUD_2569 := [[464.67, -32.7, 183.4], [0.098532, 0.700208, 0.707089, -0.005079], [0,0,0,0], [9E9, 9E9, 9E9, 9E9, 9E9, 9E9]];
	VAR robtarget OpenholeUD_2570 := [[468.64, -32.7, 183.92], [0.111226, 0.698304, 0.706865, -0.018484], [0,0,0,0], [9E9, 9E9, 9E9, 9E9, 9E9, 9E9]];
	VAR robtarget OpenholeUD_2571 := [[472.6, -32.7, 184.44], [0.123648, 0.696212, 0.706393, -0.031765], [0,0,0,0], [9E9, 9E9, 9E9, 9E9, 9E9, 9E9]];
	VAR robtarget OpenholeUD_2572 := [[476.57, -32.7, 184.96], [0.135768, 0.69395, 0.705681, -0.044883], [0,0,0,0], [9E9, 9E9, 9E9, 9E9, 9E9, 9E9]];
	VAR robtarget OpenholeUD_2573 := [[480.54, -32.7, 185.48], [0.147565, 0.691538, 0.70474, -0.057803], [0,0,0,0], [9E9, 9E9, 9E9, 9E9, 9E9, 9E9]];
	VAR robtarget OpenholeUD_2574 := [[484.5, -32.7, 186.01], [0.15902, 0.688994, 0.703584, -0.070493], [0,0,0,0], [9E9, 9E9, 9E9, 9E9, 9E9, 9E9]];
	VAR robtarget OpenholeUD_2575 := [[488.47, -32.7, 186.53], [0.170118, 0.686338, 0.702228, -0.082923], [0,0,0,0], [9E9, 9E9, 9E9, 9E9, 9E9, 9E9]];
	VAR robtarget OpenholeUD_2576 := [[492.43, -32.7, 187.05], [0.180849, 0.683589, 0.700687, -0.095069], [0,0,0,0], [9E9, 9E9, 9E9, 9E9, 9E9, 9E9]];
	VAR robtarget OpenholeUD_2577 := [[496.4, -32.7, 187.57], [0.191207, 0.680764, 0.698978, -0.106912], [0,0,0,0], [9E9, 9E9, 9E9, 9E9, 9E9, 9E9]];
	VAR robtarget OpenholeUD_2578 := [[500.36, -32.7, 188.09], [0.201187, 0.677882, 0.697118, -0.118433], [0,0,0,0], [9E9, 9E9, 9E9, 9E9, 9E9, 9E9]];
	VAR robtarget OpenholeUD_2579 := [[504.33, -32.7, 188.61], [0.21079, 0.674957, 0.695125, -0.129622], [0,0,0,0], [9E9, 9E9, 9E9, 9E9, 9E9, 9E9]];
	VAR robtarget OpenholeUD_2580 := [[509.37, -32.7, 189.28], [0.183051, 0.683002, 0.683002, -0.183051], [0,0,0,0], [9E9, 9E9, 9E9, 9E9, 9E9, 9E9]];
	VAR robtarget OpenholeUD_2581 := [[513.37, -32.7, 189.27], [0.183051, 0.683002, 0.683002, -0.183051], [0,0,0,0], [9E9, 9E9, 9E9, 9E9, 9E9, 9E9]];
	VAR robtarget OpenholeUD_2582 := [[517.37, -32.7, 189.25], [0.183051, 0.683002, 0.683002, -0.183051], [0,0,0,0], [9E9, 9E9, 9E9, 9E9, 9E9, 9E9]];
	VAR robtarget OpenholeUD_2583 := [[521.37, -32.7, 189.24], [0.183051, 0.683002, 0.683002, -0.183051], [0,0,0,0], [9E9, 9E9, 9E9, 9E9, 9E9, 9E9]];
	VAR robtarget OpenholeUD_2584 := [[529.37, -32.7, 189.22], [0.183051, 0.683002, 0.683002, -0.183051], [0,0,0,0], [9E9, 9E9, 9E9, 9E9, 9E9, 9E9]];
	VAR robtarget OpenholeUD_2585 := [[529.37, -32.7, 189.22], [0.183051, 0.683002, 0.683002, -0.183051], [0,0,0,0], [9E9, 9E9, 9E9, 9E9, 9E9, 9E9]];
	VAR robtarget OpenholeUD_2586 := [[529.37, -33.9, 189.91], [0.183051, 0.683002, 0.683002, -0.183051], [0,0,0,0], [9E9, 9E9, 9E9, 9E9, 9E9, 9E9]];
	VAR robtarget OpenholeUD_2587 := [[525.37, -33.9, 189.92], [0.183051, 0.683002, 0.683002, -0.183051], [0,0,0,0], [9E9, 9E9, 9E9, 9E9, 9E9, 9E9]];
	VAR robtarget OpenholeUD_2588 := [[521.37, -33.9, 189.93], [0.183051, 0.683002, 0.683002, -0.183051], [0,0,0,0], [9E9, 9E9, 9E9, 9E9, 9E9, 9E9]];
	VAR robtarget OpenholeUD_2589 := [[517.37, -33.9, 189.95], [0.183051, 0.683002, 0.683002, -0.183051], [0,0,0,0], [9E9, 9E9, 9E9, 9E9, 9E9, 9E9]];
	VAR robtarget OpenholeUD_2590 := [[509.37, -33.9, 189.97], [0.183051, 0.683002, 0.683002, -0.183051], [0,0,0,0], [9E9, 9E9, 9E9, 9E9, 9E9, 9E9]];
	VAR robtarget OpenholeUD_2591 := [[505.41, -33.9, 189.4], [0.216718, 0.673077, 0.695214, -0.129141], [0,0,0,0], [9E9, 9E9, 9E9, 9E9, 9E9, 9E9]];
	VAR robtarget OpenholeUD_2592 := [[501.45, -33.9, 188.84], [0.207299, 0.676038, 0.697191, -0.118], [0,0,0,0], [9E9, 9E9, 9E9, 9E9, 9E9, 9E9]];
	VAR robtarget OpenholeUD_2593 := [[497.49, -33.9, 188.27], [0.197503, 0.678964, 0.699037, -0.106526], [0,0,0,0], [9E9, 9E9, 9E9, 9E9, 9E9, 9E9]];
	VAR robtarget OpenholeUD_2594 := [[493.54, -33.9, 187.7], [0.18733, 0.681841, 0.700733, -0.094731], [0,0,0,0], [9E9, 9E9, 9E9, 9E9, 9E9, 9E9]];
	VAR robtarget OpenholeUD_2595 := [[489.58, -33.9, 187.14], [0.17678, 0.684652, 0.702262, -0.082631], [0,0,0,0], [9E9, 9E9, 9E9, 9E9, 9E9, 9E9]];
	VAR robtarget OpenholeUD_2596 := [[485.62, -33.9, 186.57], [0.165859, 0.68738, 0.703609, -0.070245], [0,0,0,0], [9E9, 9E9, 9E9, 9E9, 9E9, 9E9]];
	VAR robtarget OpenholeUD_2597 := [[481.66, -33.9, 186], [0.154577, 0.690004, 0.704757, -0.057599], [0,0,0,0], [9E9, 9E9, 9E9, 9E9, 9E9, 9E9]];
	VAR robtarget OpenholeUD_2598 := [[477.7, -33.9, 185.44], [0.142944, 0.692508, 0.705691, -0.044718], [0,0,0,0], [9E9, 9E9, 9E9, 9E9, 9E9, 9E9]];
	VAR robtarget OpenholeUD_2599 := [[473.74, -33.9, 184.87], [0.130979, 0.69487, 0.706399, -0.031635], [0,0,0,0], [9E9, 9E9, 9E9, 9E9, 9E9, 9E9]];
	VAR robtarget OpenholeUD_2600 := [[469.78, -33.9, 184.3], [0.118702, 0.697072, 0.706868, -0.018386], [0,0,0,0], [9E9, 9E9, 9E9, 9E9, 9E9, 9E9]];
	VAR robtarget OpenholeUD_2601 := [[465.82, -33.9, 183.74], [0.106139, 0.699095, 0.707089, -0.005007], [0,0,0,0], [9E9, 9E9, 9E9, 9E9, 9E9, 9E9]];
	VAR robtarget OpenholeUD_2602 := [[461.86, -33.9, 183.17], [0.09332, 0.700922, 0.707056, 0.008459], [0,0,0,0], [9E9, 9E9, 9E9, 9E9, 9E9, 9E9]];
	VAR robtarget OpenholeUD_2603 := [[457.9, -33.9, 182.61], [0.080279, 0.702535, 0.706765, 0.021971], [0,0,0,0], [9E9, 9E9, 9E9, 9E9, 9E9, 9E9]];
	VAR robtarget OpenholeUD_2604 := [[453.94, -33.9, 182.04], [0.067052, 0.70392, 0.706216, 0.035484], [0,0,0,0], [9E9, 9E9, 9E9, 9E9, 9E9, 9E9]];
	VAR robtarget OpenholeUD_2605 := [[449.98, -33.9, 181.47], [0.05368, 0.705066, 0.70541, 0.048954], [0,0,0,0], [9E9, 9E9, 9E9, 9E9, 9E9, 9E9]];
	VAR robtarget OpenholeUD_2606 := [[446.02, -33.9, 180.91], [0.040205, 0.705963, 0.704354, 0.062336], [0,0,0,0], [9E9, 9E9, 9E9, 9E9, 9E9, 9E9]];
	VAR robtarget OpenholeUD_2607 := [[442.06, -33.9, 180.34], [0.026671, 0.706604, 0.703055, 0.075589], [0,0,0,0], [9E9, 9E9, 9E9, 9E9, 9E9, 9E9]];
	VAR robtarget OpenholeUD_2608 := [[438.1, -33.9, 179.77], [0.013123, 0.706985, 0.701525, 0.088671], [0,0,0,0], [9E9, 9E9, 9E9, 9E9, 9E9, 9E9]];
	VAR robtarget OpenholeUD_2609 := [[434.14, -33.9, 179.21], [-0.000395, 0.707107, 0.699777, 0.101545], [0,0,0,0], [9E9, 9E9, 9E9, 9E9, 9E9, 9E9]];
	VAR robtarget OpenholeUD_2610 := [[430.18, -33.9, 178.64], [-0.013838, 0.706971, 0.697828, 0.114176], [0,0,0,0], [9E9, 9E9, 9E9, 9E9, 9E9, 9E9]];
	VAR robtarget OpenholeUD_2611 := [[426.22, -33.9, 178.07], [-0.027165, 0.706585, 0.695693, 0.126533], [0,0,0,0], [9E9, 9E9, 9E9, 9E9, 9E9, 9E9]];
	VAR robtarget OpenholeUD_2612 := [[422.26, -33.9, 177.51], [-0.040336, 0.705955, 0.693392, 0.138589], [0,0,0,0], [9E9, 9E9, 9E9, 9E9, 9E9, 9E9]];
	VAR robtarget OpenholeUD_2613 := [[418.3, -33.9, 176.94], [-0.053315, 0.705094, 0.690944, 0.150322], [0,0,0,0], [9E9, 9E9, 9E9, 9E9, 9E9, 9E9]];
	VAR robtarget OpenholeUD_2614 := [[414.34, -33.9, 176.37], [-0.066069, 0.704013, 0.688367, 0.161713], [0,0,0,0], [9E9, 9E9, 9E9, 9E9, 9E9, 9E9]];
	VAR robtarget OpenholeUD_2615 := [[410.38, -33.9, 175.81], [-0.078569, 0.702728, 0.685681, 0.172748], [0,0,0,0], [9E9, 9E9, 9E9, 9E9, 9E9, 9E9]];
	VAR robtarget OpenholeUD_2616 := [[406.42, -33.9, 175.24], [-0.090789, 0.701254, 0.682904, 0.183417], [0,0,0,0], [9E9, 9E9, 9E9, 9E9, 9E9, 9E9]];
	VAR robtarget OpenholeUD_2617 := [[402.46, -33.9, 174.67], [-0.102707, 0.699608, 0.680055, 0.193713], [0,0,0,0], [9E9, 9E9, 9E9, 9E9, 9E9, 9E9]];
	VAR robtarget OpenholeUD_2618 := [[398.5, -33.9, 174.11], [-0.114308, 0.697806, 0.677151, 0.203634], [0,0,0,0], [9E9, 9E9, 9E9, 9E9, 9E9, 9E9]];
	VAR robtarget OpenholeUD_2619 := [[394.54, -33.9, 173.54], [-0.125577, 0.695867, 0.674207, 0.21318], [0,0,0,0], [9E9, 9E9, 9E9, 9E9, 9E9, 9E9]];
	VAR robtarget OpenholeUD_2620 := [[389.32, -33.9, 172.79], [-0.139922, 0.693125, 0.670286, 0.225204], [0,0,0,0], [9E9, 9E9, 9E9, 9E9, 9E9, 9E9]];
	VAR robtarget OpenholeUD_2621 := [[385.32, -33.9, 172.8], [-0.183051, 0.683002, 0.683002, 0.183051], [0,0,0,0], [9E9, 9E9, 9E9, 9E9, 9E9, 9E9]];
	VAR robtarget OpenholeUD_2622 := [[381.32, -33.9, 172.82], [-0.183051, 0.683002, 0.683002, 0.183051], [0,0,0,0], [9E9, 9E9, 9E9, 9E9, 9E9, 9E9]];
	VAR robtarget OpenholeUD_2623 := [[377.32, -33.9, 172.83], [-0.183051, 0.683002, 0.683002, 0.183051], [0,0,0,0], [9E9, 9E9, 9E9, 9E9, 9E9, 9E9]];
	VAR robtarget OpenholeUD_2624 := [[373.32, -33.9, 172.84], [-0.183051, 0.683002, 0.683002, 0.183051], [0,0,0,0], [9E9, 9E9, 9E9, 9E9, 9E9, 9E9]];
	VAR robtarget OpenholeUD_2625 := [[369.32, -33.9, 172.85], [-0.183051, 0.683002, 0.683002, 0.183051], [0,0,0,0], [9E9, 9E9, 9E9, 9E9, 9E9, 9E9]];
	VAR robtarget OpenholeUD_2626 := [[369.32, -33.9, 172.85], [-0.183051, 0.683002, 0.683002, 0.183051], [0,0,0,0], [9E9, 9E9, 9E9, 9E9, 9E9, 9E9]];
	VAR robtarget OpenholeUD_2627 := [[369.32, -35.1, 172.16], [-0.183051, 0.683002, 0.683002, 0.183051], [0,0,0,0], [9E9, 9E9, 9E9, 9E9, 9E9, 9E9]];
	VAR robtarget OpenholeUD_2628 := [[373.32, -35.1, 172.15], [-0.183051, 0.683002, 0.683002, 0.183051], [0,0,0,0], [9E9, 9E9, 9E9, 9E9, 9E9, 9E9]];
	VAR robtarget OpenholeUD_2629 := [[377.32, -35.1, 172.14], [-0.183051, 0.683002, 0.683002, 0.183051], [0,0,0,0], [9E9, 9E9, 9E9, 9E9, 9E9, 9E9]];
	VAR robtarget OpenholeUD_2630 := [[381.32, -35.1, 172.12], [-0.183051, 0.683002, 0.683002, 0.183051], [0,0,0,0], [9E9, 9E9, 9E9, 9E9, 9E9, 9E9]];
	VAR robtarget OpenholeUD_2631 := [[385.32, -35.1, 172.11], [-0.183051, 0.683002, 0.683002, 0.183051], [0,0,0,0], [9E9, 9E9, 9E9, 9E9, 9E9, 9E9]];
	VAR robtarget OpenholeUD_2632 := [[389.32, -35.1, 172.1], [-0.13651, 0.693805, 0.66917, 0.228498], [0,0,0,0], [9E9, 9E9, 9E9, 9E9, 9E9, 9E9]];
	VAR robtarget OpenholeUD_2633 := [[393.27, -35.1, 172.71], [-0.125646, 0.695854, 0.672167, 0.219525], [0,0,0,0], [9E9, 9E9, 9E9, 9E9, 9E9, 9E9]];
	VAR robtarget OpenholeUD_2634 := [[397.22, -35.1, 173.32], [-0.114443, 0.697784, 0.675147, 0.210182], [0,0,0,0], [9E9, 9E9, 9E9, 9E9, 9E9, 9E9]];
	VAR robtarget OpenholeUD_2635 := [[401.18, -35.1, 173.93], [-0.102907, 0.699579, 0.678096, 0.200464], [0,0,0,0], [9E9, 9E9, 9E9, 9E9, 9E9, 9E9]];
	VAR robtarget OpenholeUD_2636 := [[405.13, -35.1, 174.54], [-0.091052, 0.70122, 0.680999, 0.190369], [0,0,0,0], [9E9, 9E9, 9E9, 9E9, 9E9, 9E9]];
	VAR robtarget OpenholeUD_2637 := [[409.08, -35.1, 175.16], [-0.078894, 0.702692, 0.683839, 0.1799], [0,0,0,0], [9E9, 9E9, 9E9, 9E9, 9E9, 9E9]];
	VAR robtarget OpenholeUD_2638 := [[413.04, -35.1, 175.77], [-0.066454, 0.703977, 0.686599, 0.16906], [0,0,0,0], [9E9, 9E9, 9E9, 9E9, 9E9, 9E9]];
	VAR robtarget OpenholeUD_2639 := [[416.99, -35.1, 176.38], [-0.053756, 0.70506, 0.689261, 0.157859], [0,0,0,0], [9E9, 9E9, 9E9, 9E9, 9E9, 9E9]];
	VAR robtarget OpenholeUD_2640 := [[420.94, -35.1, 176.99], [-0.040828, 0.705927, 0.691805, 0.146308], [0,0,0,0], [9E9, 9E9, 9E9, 9E9, 9E9, 9E9]];
	VAR robtarget OpenholeUD_2641 := [[424.89, -35.1, 177.6], [-0.027702, 0.706564, 0.694212, 0.134423], [0,0,0,0], [9E9, 9E9, 9E9, 9E9, 9E9, 9E9]];
	VAR robtarget OpenholeUD_2642 := [[428.85, -35.1, 178.21], [-0.014414, 0.70696, 0.696463, 0.122226], [0,0,0,0], [9E9, 9E9, 9E9, 9E9, 9E9, 9E9]];
	VAR robtarget OpenholeUD_2643 := [[432.8, -35.1, 178.82], [-0.001003, 0.707106, 0.698539, 0.109741], [0,0,0,0], [9E9, 9E9, 9E9, 9E9, 9E9, 9E9]];
	VAR robtarget OpenholeUD_2644 := [[436.75, -35.1, 179.43], [0.01249, 0.706996, 0.700422, 0.096997], [0,0,0,0], [9E9, 9E9, 9E9, 9E9, 9E9, 9E9]];
	VAR robtarget OpenholeUD_2645 := [[440.71, -35.1, 180.05], [0.026022, 0.706628, 0.702096, 0.084027], [0,0,0,0], [9E9, 9E9, 9E9, 9E9, 9E9, 9E9]];
	VAR robtarget OpenholeUD_2646 := [[444.66, -35.1, 180.66], [0.039548, 0.706, 0.703547, 0.070868], [0,0,0,0], [9E9, 9E9, 9E9, 9E9, 9E9, 9E9]];
	VAR robtarget OpenholeUD_2647 := [[448.61, -35.1, 181.27], [0.053024, 0.705116, 0.70476, 0.057558], [0,0,0,0], [9E9, 9E9, 9E9, 9E9, 9E9, 9E9]];
	VAR robtarget OpenholeUD_2648 := [[452.57, -35.1, 181.88], [0.066406, 0.703982, 0.705728, 0.04414], [0,0,0,0], [9E9, 9E9, 9E9, 9E9, 9E9, 9E9]];
	VAR robtarget OpenholeUD_2649 := [[456.52, -35.1, 182.49], [0.07965, 0.702606, 0.706442, 0.030657], [0,0,0,0], [9E9, 9E9, 9E9, 9E9, 9E9, 9E9]];
	VAR robtarget OpenholeUD_2650 := [[460.47, -35.1, 183.1], [0.092717, 0.701002, 0.706899, 0.017152], [0,0,0,0], [9E9, 9E9, 9E9, 9E9, 9E9, 9E9]];
	VAR robtarget OpenholeUD_2651 := [[464.42, -35.1, 183.71], [0.105568, 0.699182, 0.707097, 0.003671], [0,0,0,0], [9E9, 9E9, 9E9, 9E9, 9E9, 9E9]];
	VAR robtarget OpenholeUD_2652 := [[468.38, -35.1, 184.32], [0.118169, 0.697163, 0.70704, -0.009744], [0,0,0,0], [9E9, 9E9, 9E9, 9E9, 9E9, 9E9]];
	VAR robtarget OpenholeUD_2653 := [[472.33, -35.1, 184.94], [0.130489, 0.694962, 0.706731, -0.023051], [0,0,0,0], [9E9, 9E9, 9E9, 9E9, 9E9, 9E9]];
	VAR robtarget OpenholeUD_2654 := [[476.28, -35.1, 185.55], [0.142503, 0.692599, 0.706179, -0.03621], [0,0,0,0], [9E9, 9E9, 9E9, 9E9, 9E9, 9E9]];
	VAR robtarget OpenholeUD_2655 := [[480.24, -35.1, 186.16], [0.154187, 0.690092, 0.705394, -0.049185], [0,0,0,0], [9E9, 9E9, 9E9, 9E9, 9E9, 9E9]];
	VAR robtarget OpenholeUD_2656 := [[484.19, -35.1, 186.77], [0.165525, 0.68746, 0.704388, -0.061943], [0,0,0,0], [9E9, 9E9, 9E9, 9E9, 9E9, 9E9]];
	VAR robtarget OpenholeUD_2657 := [[488.14, -35.1, 187.38], [0.176502, 0.684724, 0.703176, -0.074454], [0,0,0,0], [9E9, 9E9, 9E9, 9E9, 9E9, 9E9]];
	VAR robtarget OpenholeUD_2658 := [[492.1, -35.1, 187.99], [0.187109, 0.681902, 0.701772, -0.086693], [0,0,0,0], [9E9, 9E9, 9E9, 9E9, 9E9, 9E9]];
	VAR robtarget OpenholeUD_2659 := [[496.05, -35.1, 188.6], [0.19734, 0.679012, 0.700193, -0.098638], [0,0,0,0], [9E9, 9E9, 9E9, 9E9, 9E9, 9E9]];
	VAR robtarget OpenholeUD_2660 := [[500, -35.1, 189.21], [0.207194, 0.67607, 0.698456, -0.110271], [0,0,0,0], [9E9, 9E9, 9E9, 9E9, 9E9, 9E9]];
	VAR robtarget OpenholeUD_2661 := [[503.95, -35.1, 189.83], [0.216669, 0.673093, 0.696576, -0.121578], [0,0,0,0], [9E9, 9E9, 9E9, 9E9, 9E9, 9E9]];
	VAR robtarget OpenholeUD_2662 := [[509.38, -35.1, 190.66], [0.183051, 0.683002, 0.683002, -0.183051], [0,0,0,0], [9E9, 9E9, 9E9, 9E9, 9E9, 9E9]];
	VAR robtarget OpenholeUD_2663 := [[513.38, -35.1, 190.65], [0.183051, 0.683002, 0.683002, -0.183051], [0,0,0,0], [9E9, 9E9, 9E9, 9E9, 9E9, 9E9]];
	VAR robtarget OpenholeUD_2664 := [[517.38, -35.1, 190.64], [0.183051, 0.683002, 0.683002, -0.183051], [0,0,0,0], [9E9, 9E9, 9E9, 9E9, 9E9, 9E9]];
	VAR robtarget OpenholeUD_2665 := [[521.38, -35.1, 190.63], [0.183051, 0.683002, 0.683002, -0.183051], [0,0,0,0], [9E9, 9E9, 9E9, 9E9, 9E9, 9E9]];
	VAR robtarget OpenholeUD_2666 := [[529.38, -35.1, 190.6], [0.183051, 0.683002, 0.683002, -0.183051], [0,0,0,0], [9E9, 9E9, 9E9, 9E9, 9E9, 9E9]];
	VAR robtarget OpenholeUD_2667 := [[529.38, -35.1, 190.6], [0.183051, 0.683002, 0.683002, -0.183051], [0,0,0,0], [9E9, 9E9, 9E9, 9E9, 9E9, 9E9]];
	VAR robtarget OpenholeUD_2668 := [[529.38, -36.3, 191.29], [0.183051, 0.683002, 0.683002, -0.183051], [0,0,0,0], [9E9, 9E9, 9E9, 9E9, 9E9, 9E9]];
	VAR robtarget OpenholeUD_2669 := [[525.38, -36.3, 191.31], [0.183051, 0.683002, 0.683002, -0.183051], [0,0,0,0], [9E9, 9E9, 9E9, 9E9, 9E9, 9E9]];
	VAR robtarget OpenholeUD_2670 := [[521.38, -36.3, 191.32], [0.183051, 0.683002, 0.683002, -0.183051], [0,0,0,0], [9E9, 9E9, 9E9, 9E9, 9E9, 9E9]];
	VAR robtarget OpenholeUD_2671 := [[517.38, -36.3, 191.33], [0.183051, 0.683002, 0.683002, -0.183051], [0,0,0,0], [9E9, 9E9, 9E9, 9E9, 9E9, 9E9]];
	VAR robtarget OpenholeUD_2672 := [[509.38, -36.3, 191.36], [0.183051, 0.683002, 0.683002, -0.183051], [0,0,0,0], [9E9, 9E9, 9E9, 9E9, 9E9, 9E9]];
	VAR robtarget OpenholeUD_2673 := [[505.43, -36.3, 190.7], [0.223455, 0.670871, 0.696458, -0.122253], [0,0,0,0], [9E9, 9E9, 9E9, 9E9, 9E9, 9E9]];
	VAR robtarget OpenholeUD_2674 := [[501.49, -36.3, 190.05], [0.214202, 0.673882, 0.698336, -0.111029], [0,0,0,0], [9E9, 9E9, 9E9, 9E9, 9E9, 9E9]];
	VAR robtarget OpenholeUD_2675 := [[497.54, -36.3, 189.39], [0.204573, 0.676868, 0.700074, -0.099479], [0,0,0,0], [9E9, 9E9, 9E9, 9E9, 9E9, 9E9]];
	VAR robtarget OpenholeUD_2676 := [[493.59, -36.3, 188.73], [0.194566, 0.679812, 0.701658, -0.087615], [0,0,0,0], [9E9, 9E9, 9E9, 9E9, 9E9, 9E9]];
	VAR robtarget OpenholeUD_2677 := [[489.65, -36.3, 188.08], [0.18418, 0.682699, 0.70307, -0.075453], [0,0,0,0], [9E9, 9E9, 9E9, 9E9, 9E9, 9E9]];
	VAR robtarget OpenholeUD_2678 := [[485.7, -36.3, 187.42], [0.173421, 0.685511, 0.704293, -0.063016], [0,0,0,0], [9E9, 9E9, 9E9, 9E9, 9E9, 9E9]];
	VAR robtarget OpenholeUD_2679 := [[481.76, -36.3, 186.77], [0.162295, 0.68823, 0.705314, -0.050326], [0,0,0,0], [9E9, 9E9, 9E9, 9E9, 9E9, 9E9]];
	VAR robtarget OpenholeUD_2680 := [[477.81, -36.3, 186.11], [0.150814, 0.690837, 0.706116, -0.037413], [0,0,0,0], [9E9, 9E9, 9E9, 9E9, 9E9, 9E9]];
	VAR robtarget OpenholeUD_2681 := [[473.87, -36.3, 185.46], [0.138993, 0.693312, 0.706689, -0.024308], [0,0,0,0], [9E9, 9E9, 9E9, 9E9, 9E9, 9E9]];
	VAR robtarget OpenholeUD_2682 := [[469.92, -36.3, 184.8], [0.126853, 0.695635, 0.70702, -0.011047], [0,0,0,0], [9E9, 9E9, 9E9, 9E9, 9E9, 9E9]];
	VAR robtarget OpenholeUD_2683 := [[465.97, -36.3, 184.14], [0.114417, 0.697788, 0.707103, 0.002331], [0,0,0,0], [9E9, 9E9, 9E9, 9E9, 9E9, 9E9]];
	VAR robtarget OpenholeUD_2684 := [[462.03, -36.3, 183.49], [0.101714, 0.699753, 0.706931, 0.015786], [0,0,0,0], [9E9, 9E9, 9E9, 9E9, 9E9, 9E9]];
	VAR robtarget OpenholeUD_2685 := [[458.08, -36.3, 182.83], [0.088777, 0.701512, 0.706501, 0.029274], [0,0,0,0], [9E9, 9E9, 9E9, 9E9, 9E9, 9E9]];
	VAR robtarget OpenholeUD_2686 := [[454.14, -36.3, 182.18], [0.07564, 0.703049, 0.705813, 0.042752], [0,0,0,0], [9E9, 9E9, 9E9, 9E9, 9E9, 9E9]];
	VAR robtarget OpenholeUD_2687 := [[450.19, -36.3, 181.52], [0.062344, 0.704353, 0.704872, 0.056176], [0,0,0,0], [9E9, 9E9, 9E9, 9E9, 9E9, 9E9]];
	VAR robtarget OpenholeUD_2688 := [[446.24, -36.3, 180.87], [0.04893, 0.705412, 0.703683, 0.069501], [0,0,0,0], [9E9, 9E9, 9E9, 9E9, 9E9, 9E9]];
	VAR robtarget OpenholeUD_2689 := [[442.3, -36.3, 180.21], [0.035441, 0.706218, 0.702255, 0.082687], [0,0,0,0], [9E9, 9E9, 9E9, 9E9, 9E9, 9E9]];
	VAR robtarget OpenholeUD_2690 := [[438.35, -36.3, 179.55], [0.021922, 0.706767, 0.700602, 0.095694], [0,0,0,0], [9E9, 9E9, 9E9, 9E9, 9E9, 9E9]];
	VAR robtarget OpenholeUD_2691 := [[434.41, -36.3, 178.9], [0.008417, 0.707057, 0.698736, 0.108483], [0,0,0,0], [9E9, 9E9, 9E9, 9E9, 9E9, 9E9]];
	VAR robtarget OpenholeUD_2692 := [[430.46, -36.3, 178.24], [-0.005031, 0.707089, 0.696674, 0.121021], [0,0,0,0], [9E9, 9E9, 9E9, 9E9, 9E9, 9E9]];
	VAR robtarget OpenholeUD_2693 := [[426.51, -36.3, 177.59], [-0.018378, 0.706868, 0.694433, 0.133277], [0,0,0,0], [9E9, 9E9, 9E9, 9E9, 9E9, 9E9]];
	VAR robtarget OpenholeUD_2694 := [[422.57, -36.3, 176.93], [-0.031584, 0.706401, 0.692032, 0.145227], [0,0,0,0], [9E9, 9E9, 9E9, 9E9, 9E9, 9E9]];
	VAR robtarget OpenholeUD_2695 := [[418.62, -36.3, 176.28], [-0.044614, 0.705698, 0.689491, 0.156849], [0,0,0,0], [9E9, 9E9, 9E9, 9E9, 9E9, 9E9]];
	VAR robtarget OpenholeUD_2696 := [[414.68, -36.3, 175.62], [-0.057432, 0.704771, 0.686829, 0.168124], [0,0,0,0], [9E9, 9E9, 9E9, 9E9, 9E9, 9E9]];
	VAR robtarget OpenholeUD_2697 := [[410.73, -36.3, 174.96], [-0.070009, 0.703633, 0.684065, 0.17904], [0,0,0,0], [9E9, 9E9, 9E9, 9E9, 9E9, 9E9]];
	VAR robtarget OpenholeUD_2698 := [[406.78, -36.3, 174.31], [-0.082317, 0.702299, 0.681217, 0.189587], [0,0,0,0], [9E9, 9E9, 9E9, 9E9, 9E9, 9E9]];
	VAR robtarget OpenholeUD_2699 := [[402.84, -36.3, 173.65], [-0.094336, 0.700786, 0.678304, 0.199759], [0,0,0,0], [9E9, 9E9, 9E9, 9E9, 9E9, 9E9]];
	VAR robtarget OpenholeUD_2700 := [[398.89, -36.3, 173], [-0.106045, 0.69911, 0.675342, 0.209555], [0,0,0,0], [9E9, 9E9, 9E9, 9E9, 9E9, 9E9]];
	VAR robtarget OpenholeUD_2701 := [[394.95, -36.3, 172.34], [-0.117431, 0.697288, 0.672346, 0.218975], [0,0,0,0], [9E9, 9E9, 9E9, 9E9, 9E9, 9E9]];
	VAR robtarget OpenholeUD_2702 := [[389.31, -36.3, 171.41], [-0.133103, 0.694466, 0.668041, 0.231777], [0,0,0,0], [9E9, 9E9, 9E9, 9E9, 9E9, 9E9]];
	VAR robtarget OpenholeUD_2703 := [[385.31, -36.3, 171.42], [-0.183051, 0.683002, 0.683002, 0.183051], [0,0,0,0], [9E9, 9E9, 9E9, 9E9, 9E9, 9E9]];
	VAR robtarget OpenholeUD_2704 := [[381.31, -36.3, 171.43], [-0.183051, 0.683002, 0.683002, 0.183051], [0,0,0,0], [9E9, 9E9, 9E9, 9E9, 9E9, 9E9]];
	VAR robtarget OpenholeUD_2705 := [[377.31, -36.3, 171.44], [-0.183051, 0.683002, 0.683002, 0.183051], [0,0,0,0], [9E9, 9E9, 9E9, 9E9, 9E9, 9E9]];
	VAR robtarget OpenholeUD_2706 := [[373.31, -36.3, 171.46], [-0.183051, 0.683002, 0.683002, 0.183051], [0,0,0,0], [9E9, 9E9, 9E9, 9E9, 9E9, 9E9]];
	VAR robtarget OpenholeUD_2707 := [[369.31, -36.3, 171.47], [-0.183051, 0.683002, 0.683002, 0.183051], [0,0,0,0], [9E9, 9E9, 9E9, 9E9, 9E9, 9E9]];
	VAR robtarget OpenholeUD_2708 := [[369.31, -36.3, 171.47], [-0.183051, 0.683002, 0.683002, 0.183051], [0,0,0,0], [9E9, 9E9, 9E9, 9E9, 9E9, 9E9]];
	VAR robtarget OpenholeUD_2709 := [[369.31, -37.5, 170.78], [-0.183051, 0.683002, 0.683002, 0.183051], [0,0,0,0], [9E9, 9E9, 9E9, 9E9, 9E9, 9E9]];
	VAR robtarget OpenholeUD_2710 := [[373.31, -37.5, 170.76], [-0.183051, 0.683002, 0.683002, 0.183051], [0,0,0,0], [9E9, 9E9, 9E9, 9E9, 9E9, 9E9]];
	VAR robtarget OpenholeUD_2711 := [[377.31, -37.5, 170.75], [-0.183051, 0.683002, 0.683002, 0.183051], [0,0,0,0], [9E9, 9E9, 9E9, 9E9, 9E9, 9E9]];
	VAR robtarget OpenholeUD_2712 := [[381.31, -37.5, 170.74], [-0.183051, 0.683002, 0.683002, 0.183051], [0,0,0,0], [9E9, 9E9, 9E9, 9E9, 9E9, 9E9]];
	VAR robtarget OpenholeUD_2713 := [[385.31, -37.5, 170.73], [-0.183051, 0.683002, 0.683002, 0.183051], [0,0,0,0], [9E9, 9E9, 9E9, 9E9, 9E9, 9E9]];
	VAR robtarget OpenholeUD_2714 := [[389.31, -37.5, 170.71], [-0.129702, 0.69511, 0.6669, 0.235042], [0,0,0,0], [9E9, 9E9, 9E9, 9E9, 9E9, 9E9]];
	VAR robtarget OpenholeUD_2715 := [[393.25, -37.5, 171.41], [-0.118755, 0.697063, 0.669939, 0.226235], [0,0,0,0], [9E9, 9E9, 9E9, 9E9, 9E9, 9E9]];
	VAR robtarget OpenholeUD_2716 := [[397.19, -37.5, 172.11], [-0.107472, 0.698892, 0.672968, 0.217059], [0,0,0,0], [9E9, 9E9, 9E9, 9E9, 9E9, 9E9]];
	VAR robtarget OpenholeUD_2717 := [[401.13, -37.5, 172.81], [-0.095865, 0.700578, 0.675974, 0.207508], [0,0,0,0], [9E9, 9E9, 9E9, 9E9, 9E9, 9E9]];
	VAR robtarget OpenholeUD_2718 := [[405.07, -37.5, 173.51], [-0.083945, 0.702106, 0.678942, 0.197579], [0,0,0,0], [9E9, 9E9, 9E9, 9E9, 9E9, 9E9]];
	VAR robtarget OpenholeUD_2719 := [[409, -37.5, 174.21], [-0.071731, 0.703459, 0.681856, 0.187275], [0,0,0,0], [9E9, 9E9, 9E9, 9E9, 9E9, 9E9]];
	VAR robtarget OpenholeUD_2720 := [[412.94, -37.5, 174.91], [-0.059244, 0.704621, 0.684699, 0.176597], [0,0,0,0], [9E9, 9E9, 9E9, 9E9, 9E9, 9E9]];
	VAR robtarget OpenholeUD_2721 := [[416.88, -37.5, 175.61], [-0.046508, 0.705576, 0.687453, 0.165554], [0,0,0,0], [9E9, 9E9, 9E9, 9E9, 9E9, 9E9]];
	VAR robtarget OpenholeUD_2722 := [[420.82, -37.5, 176.31], [-0.033552, 0.70631, 0.690098, 0.154156], [0,0,0,0], [9E9, 9E9, 9E9, 9E9, 9E9, 9E9]];
	VAR robtarget OpenholeUD_2723 := [[424.76, -37.5, 177.01], [-0.02041, 0.706812, 0.692616, 0.142418], [0,0,0,0], [9E9, 9E9, 9E9, 9E9, 9E9, 9E9]];
	VAR robtarget OpenholeUD_2724 := [[428.7, -37.5, 177.71], [-0.007116, 0.707071, 0.694987, 0.130359], [0,0,0,0], [9E9, 9E9, 9E9, 9E9, 9E9, 9E9]];
	VAR robtarget OpenholeUD_2725 := [[432.63, -37.5, 178.41], [0.006289, 0.707079, 0.697191, 0.118004], [0,0,0,0], [9E9, 9E9, 9E9, 9E9, 9E9, 9E9]];
	VAR robtarget OpenholeUD_2726 := [[436.57, -37.5, 179.11], [0.019765, 0.70683, 0.699211, 0.105378], [0,0,0,0], [9E9, 9E9, 9E9, 9E9, 9E9, 9E9]];
	VAR robtarget OpenholeUD_2727 := [[440.51, -37.5, 179.81], [0.033269, 0.706324, 0.701028, 0.092515], [0,0,0,0], [9E9, 9E9, 9E9, 9E9, 9E9, 9E9]];
	VAR robtarget OpenholeUD_2728 := [[444.45, -37.5, 180.51], [0.046755, 0.705559, 0.702629, 0.079449], [0,0,0,0], [9E9, 9E9, 9E9, 9E9, 9E9, 9E9]];
	VAR robtarget OpenholeUD_2729 := [[448.39, -37.5, 181.21], [0.060181, 0.704541, 0.703999, 0.066219], [0,0,0,0], [9E9, 9E9, 9E9, 9E9, 9E9, 9E9]];
	VAR robtarget OpenholeUD_2730 := [[452.33, -37.5, 181.91], [0.073501, 0.703276, 0.705128, 0.052865], [0,0,0,0], [9E9, 9E9, 9E9, 9E9, 9E9, 9E9]];
	VAR robtarget OpenholeUD_2731 := [[456.26, -37.5, 182.61], [0.086675, 0.701774, 0.706007, 0.039431], [0,0,0,0], [9E9, 9E9, 9E9, 9E9, 9E9, 9E9]];
	VAR robtarget OpenholeUD_2732 := [[460.2, -37.5, 183.31], [0.099662, 0.700048, 0.70663, 0.02596], [0,0,0,0], [9E9, 9E9, 9E9, 9E9, 9E9, 9E9]];
	VAR robtarget OpenholeUD_2733 := [[464.14, -37.5, 184.01], [0.112425, 0.698112, 0.706996, 0.012495], [0,0,0,0], [9E9, 9E9, 9E9, 9E9, 9E9, 9E9]];
	VAR robtarget OpenholeUD_2734 := [[468.08, -37.5, 184.71], [0.124931, 0.695983, 0.707106, -0.000919], [0,0,0,0], [9E9, 9E9, 9E9, 9E9, 9E9, 9E9]];
	VAR robtarget OpenholeUD_2735 := [[472.02, -37.5, 185.41], [0.13715, 0.693679, 0.706963, -0.014241], [0,0,0,0], [9E9, 9E9, 9E9, 9E9, 9E9, 9E9]];
	VAR robtarget OpenholeUD_2736 := [[475.96, -37.5, 186.11], [0.149056, 0.691218, 0.706574, -0.027432], [0,0,0,0], [9E9, 9E9, 9E9, 9E9, 9E9, 9E9]];
	VAR robtarget OpenholeUD_2737 := [[479.89, -37.5, 186.81], [0.160628, 0.688621, 0.705949, -0.040452], [0,0,0,0], [9E9, 9E9, 9E9, 9E9, 9E9, 9E9]];
	VAR robtarget OpenholeUD_2738 := [[483.83, -37.5, 187.51], [0.17185, 0.685907, 0.705097, -0.05327], [0,0,0,0], [9E9, 9E9, 9E9, 9E9, 9E9, 9E9]];
	VAR robtarget OpenholeUD_2739 := [[487.77, -37.5, 188.21], [0.182707, 0.683094, 0.704034, -0.065854], [0,0,0,0], [9E9, 9E9, 9E9, 9E9, 9E9, 9E9]];
	VAR robtarget OpenholeUD_2740 := [[491.71, -37.5, 188.91], [0.193193, 0.680203, 0.702772, -0.078177], [0,0,0,0], [9E9, 9E9, 9E9, 9E9, 9E9, 9E9]];
